(*=======================================================*)
	110: (* WT-Abfrage auf Beladeposition *)

		IF NOT e_station_vorher_in_abgegeben THEN
			a_station_vorher_out_angekommen := FALSE;
			bm_abfrage_wt_auf_beladepos := TRUE;
		END_IF

		(*-----------------------Weiterschaltbedingungen----------------------------*)
		IF e_wt_auf_beladepos THEN
			(* Ein WT ist anwesend zum rausschicken *)
			IF NOT ST_WT_Transport_Abgabe.e_wt_auf_abgabepos THEN
				(* Erst wenn kein Stau vorhanden ist, dann wird der WT weiter gelassen *)
				fb_state_entry.i16_next_step := 120;
			END_IF
		ELSE
			fb_state_entry.i16_next_step := 140;
		END_IF

		IF fb_state_entry.X THEN
			bm_abfrage_wt_auf_beladepos := FALSE;
			st_ctrl_out.b_kontroller_start := FALSE;
		END_IF

(*=======================================================*)
	120: (* WT-Zentrierer und Stopper einfahren *)
		IF fb_state_entry.E THEN
			zyl_wt_stopper_tisch.st_ctrl.in.b_einfahren := TRUE;
			zyl_wt_zentrierer_tisch.st_ctrl.in.b_einfahren := TRUE;
			fb_Zentrierer_einfahren(b_start:= TRUE, t_zeit=> );
			fb_Tisch_WechselZeit(b_start:=TRUE , t_zeit=> );
			pm_traegerwechselzeit := FALSE;
		END_IF

		IF 	zyl_wt_zentrierer_tisch.st_ctrl.out.b_eingefahren THEN
			fb_Zentrierer_einfahren(b_start:= FALSE, t_zeit=>t_Zentrierer_einfahren );
		END_IF

		(*-----------------------Weiterschaltbedingungen----------------------------*)
		IF zyl_wt_stopper_tisch.st_ctrl.out.b_eingefahren AND zyl_wt_zentrierer_tisch.st_ctrl.out.b_eingefahren THEN
			zyl_wt_stopper_tisch.st_ctrl.in.b_einfahren := FALSE;
			zyl_wt_zentrierer_tisch.st_ctrl.in.b_einfahren := FALSE;
			fb_state_entry.i16_next_step := 130;
		END_IF

(*=======================================================*)
	130: (* WT fährt von Bestücktisch heraus *)
		IF fb_state_entry.E THEN
			fb_ton_uez.PT := t#5s;
 			fb_ton_uez.IN := TRUE;
			st_ctrl_out.b_kontroller_start := TRUE;
		END_IF

		(*-----------------------Weiterschaltbedingungen----------------------------*)
		IF fb_r_trig_beladepos_verlassen.Q THEN
			fb_ton_uez.IN := FALSE;
			st_ctrl_out.b_kontroller_start := FALSE;
			IF	gst_datensatz.st_md.i16_WdhTouchProbe = 0 THEN
				fb_state_entry.i16_next_step := 144;
			ELSE
				fb_state_entry.i16_next_step := 140;
			END_IF
		ELSIF fb_ton_uez.Q THEN
			sm_wt_hat_beladepos_nicht_verlassen := TRUE;
			fb_state_entry.i16_next_step := FEHLER;
		END_IF

(*=======================================================*)
	140: (* Starte Touchprobe => kann immer gestartet werden. Wenn kein Taster eingebaut ist, wird gleich wieder fertig gemeldet*)
		IF fb_state_entry.E THEN
			ST_TouchProbe.st_ctrl_in.b_start := TRUE;
		END_IF

		(*-----------------------Weiterschaltbedingungen----------------------------*)
		IF	ST_TouchProbe.st_ctrl_out.b_busy THEN
			fb_state_entry.i16_next_step := 142;
		END_IF

(*=======================================================*)
	142: (* Warte auf fertig*)

		(*-----------------------Weiterschaltbedingungen----------------------------*)
		IF	ST_TouchProbe.st_ctrl_out.b_fertig THEN
			fb_state_entry.i16_next_step := 144;
		END_IF

(*=======================================================*)
	144: (* Stopper in Simulation nicht ausfahren  und  WT-Zentrierer einfahren *)
		IF fb_state_entry.E THEN
			zyl_wt_stopper_tisch.st_ctrl.in.b_ausfahren := TRUE;
			zyl_wt_zentrierer_tisch.st_ctrl.in.b_einfahren := TRUE;
		END_IF

		(*-----------------------Weiterschaltbedingungen----------------------------*)
		IF 	zyl_wt_stopper_tisch.st_ctrl.out.b_ausgefahren AND
			zyl_wt_zentrierer_tisch.st_ctrl.out.b_eingefahren
			THEN
				zyl_wt_stopper_tisch.st_ctrl.in.b_ausfahren := FALSE;
				zyl_wt_zentrierer_tisch.st_ctrl.in.b_einfahren := FALSE;
				fb_Tisch_WechselZeit(b_start:=FALSE , t_zeit=>t_tischwechselzeit );
				pm_traegerwechselzeit := t_tischwechselzeit > gst_datensatz.st_md.t_max_tischwechselzeit AND gst_datensatz.st_md.t_max_tischwechselzeit <> INT_TO_TIME(0);
				fb_state_entry.i16_next_step := 150;
		END_IF

(*=======================================================*)
	150: (* Warte auf Anforderung von vorheriger Station *)
		IF fb_state_entry.E THEN
			bm_warte_anforderung := TRUE;
		END_IF

		(*-----------------------Weiterschaltbedingungen----------------------------*)
		IF e_station_vorher_in_anforderung AND NOT e_wt_auf_beladepos THEN
			a_station_vorher_out_angekommen := FALSE;
			a_station_vorher_out_erlaubnis := TRUE;
			st_ctrl_out.b_kontroller_start := TRUE;
			bm_warte_anforderung := FALSE;
			fb_state_entry.i16_next_step := 160;
		END_IF

(*=======================================================*)
	160: (* Warte bis angekommen an Tisch-Stopper *)
		IF fb_state_entry.E THEN
			bm_warte_auf_wt_an_stopper := TRUE;
		END_IF

		IF e_wt_im_aktionsfeld AND NOT fb_ton_wz.Q THEN
			fb_ton_wz.PT := t#3s;
			fb_ton_wz.IN := TRUE;
		END_IF

		(*Kontroller neu starten wenn das Förderband zwischenzeitlich abgeschaltet hat*)
		IF 	e_station_vorher_in_abgegeben AND NOT ST_WT_Transport_Kontroller.a_foerderband_wt_transport THEN
			st_ctrl_out.b_kontroller_start := TRUE;
		ELSE
			st_ctrl_out.b_kontroller_start := FALSE;
		END_IF

		(*-----------------------Weiterschaltbedingungen----------------------------*)
		(* Auf das Kommando "e_station_vorher_in_abgegeben" wird nicht gewartet,
		da auch mal ein WT nach einer Störung so aus der vorherigen Station kommen kann. *)
		IF fb_ton_wt_auf_beladepos.Q THEN
			st_ctrl_out.b_kontroller_start := FALSE;
			a_station_vorher_out_erlaubnis := FALSE;
			a_station_vorher_out_angekommen := TRUE;
			bm_warte_auf_wt_an_stopper := FALSE;
			fb_ton_wz.IN := FALSE;
			fb_state_entry.i16_next_step := 170;
		END_IF

		(*Abfrage auf Sensorfehler des Beladepositionssensors *)
		IF e_wt_im_aktionsfeld AND NOT e_wt_auf_beladepos AND fb_ton_wz.Q THEN
			sm_sensorfehler_beladepos := TRUE;
			fb_state_entry.i16_next_step := FEHLER;
		END_IF

(*=======================================================*)
	170: (* WT-Zentrierer ausfahren *)
		IF fb_state_entry.E THEN
			zyl_wt_zentrierer_tisch.st_ctrl.in.b_ausfahren := TRUE;
			fb_Zentrierer_ausfahren(b_start:= TRUE, t_zeit=> );
		END_IF

		(*-----------------------Weiterschaltbedingungen----------------------------*)
		IF zyl_wt_zentrierer_tisch.st_ctrl.out.b_ausgefahren AND
			NOT ST_TippTasten.b_einfaedeln_aktiv AND
			(NOT ST_Virtuelle_Masterachse.b_merker_bandende_links  OR
 			NOT ST_Virtuelle_Masterachse.b_merker_bandende_rechts) THEN
			zyl_wt_zentrierer_tisch.st_ctrl.in.b_ausfahren := FALSE;
			fb_Zentrierer_ausfahren(b_start:= FALSE, t_zeit=> t_Zentrierer_ausfahren);
			zyl_wt_zentrierer_tisch.st_ctrl.in.b_ausfahren := FALSE;
			IF st_config.b_station_in_simulation THEN
				(* WT-Transport ist in Simulation und deshalb wird der WT ohne zu Bestücken weiter gefahren *)
				fb_state_entry.i16_next_step := BEREIT;
			ELSE
				fb_state_entry.i16_next_step := 190;
			END_IF
		END_IF

(*=======================================================*)
	190: (* WT-Tag mit RFID-Lesegerät abfragen *)
		IF fb_state_entry.E THEN
			fb_ton_wz.PT := t#100ms;
			fb_ton_wz.IN := TRUE;
		END_IF

		(*-----------------------Weiterschaltbedingungen----------------------------*)
		IF fb_ton_wz.Q THEN
			IF e_wt_im_aktionsfeld THEN
				(* Tag auslesen *)
				fb_state_entry.i16_next_step := 240;
			ELSE
				(* Kein Tag auf WT *)
				sm_wt_hat_kein_tag := TRUE;
				fb_state_entry.i16_next_step := FEHLER;
			END_IF
		END_IF

		IF fb_state_entry.X THEN
			fb_ton_wz.IN := FALSE;
		END_IF

(*=======================================================*)
	240: (* Starte Z-Achse *)
		IF fb_state_entry.E THEN
			axis_z_achse.st_ctrl.in.b_start := TRUE;
			st_ctrl_out.b_kontroller_start := TRUE;
			(*Zeitmessung Trägerwechsel stoppen und ausgeben*)
			fb_WT_WechselZeit(b_start:=FALSE , t_zeit=>t_WT_WechselZeit );
			(*Zeitmessung Bestückvorgang starten*)
			fb_Zentrierer_ausfahren(b_start:= FALSE, t_zeit=>t_Zentrierer_ausfahren );
		END_IF

		(*-----------------------Weiterschaltbedingungen----------------------------*)
		IF axis_z_achse.st_ctrl.out.b_fertig AND NOT fb_state_entry.E THEN
			axis_z_achse.st_ctrl.in.b_start := FALSE;
			st_ctrl_out.b_kontroller_start := FALSE;
			stueckzahlen.st_ctrl.in.b_gutteil_produziert := TRUE;
			(*Zeitmessung Trägerwechsel starten*)
			fb_WT_WechselZeit(b_start:=TRUE , t_zeit=> );
			(*Zeitmessung zusammenfassen*)
			t_bestueckzeit:=ST_Z_Achse.t_Bestueckung;
			t_traegerwechselzeit:=t_WT_WechselZeit + ST_Z_Achse.t_Z_Achse_einfahren + ST_Z_Achse.t_Z_Achse_ausfahren;
			t_komplett_zyklus:= t_traegerwechselzeit + t_bestueckzeit;
			fb_state_entry.i16_next_step := BEREIT;
		END_IF

		IF fb_state_entry.X THEN
			gst_datensatz.st_md.produzierte_Stecker := gst_datensatz.st_md.produzierte_Stecker + 1;
		END_IF

(*=======================================================*)
	500: (* Warte bis angekommen an Stopper *)
		IF fb_state_entry.E THEN
			bm_warte_auf_wt_an_stopper := TRUE;
		END_IF

		IF e_wt_im_aktionsfeld AND NOT fb_ton_wz.Q THEN
			fb_ton_wz.PT := t#3s;
			fb_ton_wz.IN := TRUE;
		END_IF

		(*-----------------------Weiterschaltbedingungen----------------------------*)
		IF fb_ton_wt_auf_beladepos.Q THEN
			fb_ton_wz.IN := FALSE;
			fb_state_entry.i16_next_step := 510;
		END_IF

		(*Abfrage auf Sensorfehler des Beladepositionssensors *)
		IF e_wt_im_aktionsfeld AND NOT e_wt_auf_beladepos AND fb_ton_wz.Q THEN
			sm_sensorfehler_beladepos := TRUE;
			fb_state_entry.i16_next_step := FEHLER;
		END_IF

(*=======================================================*)
	510: (* WT-Zentrierer ausfahren *)
		IF fb_state_entry.E THEN
			zyl_wt_zentrierer_tisch.st_ctrl.in.b_ausfahren := TRUE;
		END_IF

		(*-----------------------Weiterschaltbedingungen----------------------------*)
		IF zyl_wt_zentrierer_tisch.st_ctrl.out.b_ausgefahren  THEN
			zyl_wt_zentrierer_tisch.st_ctrl.in.b_ausfahren := FALSE;
			fb_state_entry.i16_next_step := 520;
		END_IF

(*=======================================================*)
	520:	(* Produktion ohne aktiven WT Transport *)
		IF fb_state_entry.E THEN
			axis_z_achse.st_ctrl.in.b_start := TRUE;
		END_IF

		(*-----------------------Weiterschaltbedingungen----------------------------*)
		IF axis_z_achse.st_ctrl.out.b_fertig AND NOT fb_state_entry.E THEN
			axis_z_achse.st_ctrl.in.b_start := FALSE;
			stueckzahlen.st_ctrl.in.b_gutteil_produziert := TRUE;
			IF NOT b_Dauertest_Achsen THEN
				fb_state_entry.i16_next_step := BEREIT;
			ELSE
				(* zum Testen der Achsen nach Tausch, Bestückbild "Becherspucken", WKZ ausgebaut, Vorschubkontrolle abeschaltet,
				Bit muss von Programmierer geforct werden, zum Beenden Schlüsselschalter auf HAND und Zelle neu starten *)
				fb_state_entry.i16_next_step := 500;	(* Dauertest *)
			END_IF
		END_IF

		IF fb_state_entry.X AND NOT b_Dauertest_Achsen THEN
			gst_datensatz.st_md.produzierte_Stecker := gst_datensatz.st_md.produzierte_Stecker + 1;
		END_IF

(*=======================================================*)
	FEHLER:
		IF fb_state_entry.E THEN
			st_ctrl_out.b_fehler := TRUE;
			fb_ton_quitt.IN := FALSE;
			zyl_wt_zentrierer_tisch.st_ctrl.in.b_quittieren := FALSE;
			zyl_wt_stopper_tisch.st_ctrl.in.b_quittieren := FALSE;

			a_station_vorher_out_erlaubnis := FALSE;
			a_station_vorher_out_angekommen := FALSE;

			st_ctrl_out.b_kontroller_start := FALSE;

			(*ST_Markiere_WT_NIO();*)
		END_IF

		(*-----------------------Weiterschaltbedingungen----------------------------*)
		IF st_ctrl_in.b_quitt AND NOT fb_state_entry.E THEN
			st_ctrl_out.b_fehler := FALSE;
			zyl_wt_zentrierer_tisch.st_ctrl.in.b_quittieren := TRUE;
			zyl_wt_stopper_tisch.st_ctrl.in.b_quittieren := TRUE;
			fb_ton_quitt.IN := TRUE;
		END_IF

		IF fb_ton_quitt.Q THEN
			fb_ton_quitt.IN := FALSE;
			fb_state_entry.i16_next_step := INIT;
		END_IF

(*=======================================================*)
	STOP:
		IF fb_state_entry.E THEN
			fb_ton_quitt.IN := FALSE;
			st_ctrl_out.b_kontroller_start := FALSE;
			zyl_wt_zentrierer_tisch.st_ctrl.in.b_quittieren := FALSE;
			zyl_wt_stopper_tisch.st_ctrl.in.b_quittieren := FALSE;
			a_station_vorher_out_erlaubnis := FALSE;
			a_station_vorher_out_angekommen := FALSE;
			(*ST_Markiere_WT_NIO();*)
		END_IF

		(*-----------------------Weiterschaltbedingungen----------------------------*)
		IF st_ctrl_in.b_quitt AND NOT fb_state_entry.E THEN
			fb_ton_quitt.IN := TRUE;
			zyl_wt_zentrierer_tisch.st_ctrl.in.b_quittieren := TRUE;
			zyl_wt_stopper_tisch.st_ctrl.in.b_quittieren := TRUE;
		END_IF

		IF fb_ton_quitt.Q THEN
			fb_ton_quitt.IN := FALSE;
			fb_state_entry.i16_next_step := INIT;
		END_IF
END_CASE

fb_state_entry(
	i16_next_step:= ,
	i16_pos:= 2,
	s_debugtext:= ,
	E=> ,
	X=> ,
	i16_step=> ,
	i16_last_step=> );

fb_ton_abfrage_wt_auf_beladepos (IN:=bm_abfrage_wt_auf_beladepos,PT:=t#30s);
fb_ton_warte_anforderung (IN:=bm_warte_anforderung,PT:=t#30s);
fb_ton_warte_auf_wt_an_stopper (IN:=bm_warte_auf_wt_an_stopper,PT:=t#30s);

IF st_config.b_config_fertig THEN
	(* Fehlermeldungen ab dem Startindex in das globale Störmeldungsarray schreiben *)
	garr_stoermeldungen[st_config.i16_meld_startindex + 0] := sm_wt_hat_beladepos_nicht_verlassen;
	garr_stoermeldungen[st_config.i16_meld_startindex + 1] := sm_tagnummer_ungueltig;
	garr_stoermeldungen[st_config.i16_meld_startindex + 2] := sm_wt_hat_kein_tag;
	garr_stoermeldungen[st_config.i16_meld_startindex + 3] := FALSE;
	garr_stoermeldungen[st_config.i16_meld_startindex + 4] := sm_sensorfehler_beladepos;
	garr_stoermeldungen[st_config.i16_meld_startindex + 5] := sm_tagreader_nicht_fertig;
	garr_stoermeldungen[st_config.i16_meld_startindex + 6] := sm_wt_zu_frueh_in_zelle;
	garr_stoermeldungen[st_config.i16_meld_startindex + 7] := sm_keine_bandfreigabe;
	garr_stoermeldungen[st_config.i16_meld_startindex + 8] := FALSE;
	garr_stoermeldungen[st_config.i16_meld_startindex + 9] := FALSE;
	garr_stoermeldungen[st_config.i16_meld_startindex + 10] := FALSE;
	garr_stoermeldungen[st_config.i16_meld_startindex + 11] := FALSE;
	garr_stoermeldungen[st_config.i16_meld_startindex + 12] := FALSE;
	garr_stoermeldungen[st_config.i16_meld_startindex + 13] := FALSE;
	garr_stoermeldungen[st_config.i16_meld_startindex + 14] := FALSE;
	garr_stoermeldungen[st_config.i16_meld_startindex + 15] := FALSE;
	garr_stoermeldungen[st_config.i16_meld_startindex + 16] := FALSE;
	garr_stoermeldungen[st_config.i16_meld_startindex + 17] := FALSE;
	garr_stoermeldungen[st_config.i16_meld_startindex + 18] := FALSE;
	garr_stoermeldungen[st_config.i16_meld_startindex + 19] := FALSE;
	
	garr_betriebsmeldungen[st_config.i16_meld_startindex + 0] := fb_ton_abfrage_wt_auf_beladepos.Q;
	garr_betriebsmeldungen[st_config.i16_meld_startindex + 1] := fb_ton_warte_anforderung.Q;
	garr_betriebsmeldungen[st_config.i16_meld_startindex + 2] := fb_ton_warte_auf_wt_an_stopper.Q;
	garr_betriebsmeldungen[st_config.i16_meld_startindex + 3] := FALSE;
	garr_betriebsmeldungen[st_config.i16_meld_startindex + 4] := FALSE;
	garr_betriebsmeldungen[st_config.i16_meld_startindex + 5] := FALSE;
	garr_betriebsmeldungen[st_config.i16_meld_startindex + 6] := FALSE;
	garr_betriebsmeldungen[st_config.i16_meld_startindex + 7] := FALSE;
	garr_betriebsmeldungen[st_config.i16_meld_startindex + 8] := FALSE;
	garr_betriebsmeldungen[st_config.i16_meld_startindex + 9] := FALSE;
	garr_betriebsmeldungen[st_config.i16_meld_startindex + 10] := FALSE;
	garr_betriebsmeldungen[st_config.i16_meld_startindex + 11] := FALSE;
	garr_betriebsmeldungen[st_config.i16_meld_startindex + 12] := FALSE;
	garr_betriebsmeldungen[st_config.i16_meld_startindex + 13] := FALSE;
	garr_betriebsmeldungen[st_config.i16_meld_startindex + 14] := FALSE;
	garr_betriebsmeldungen[st_config.i16_meld_startindex + 15] := FALSE;
	garr_betriebsmeldungen[st_config.i16_meld_startindex + 16] := FALSE;
	garr_betriebsmeldungen[st_config.i16_meld_startindex + 17] := FALSE;
	garr_betriebsmeldungen[st_config.i16_meld_startindex + 18] := FALSE;
	garr_betriebsmeldungen[st_config.i16_meld_startindex + 19] := FALSE;
END_IF
END_PROGRAM

(* POU Gemeinsamkeiten17xx/WT Transport/ST_WT_Transport_Kontroller, ST *)
PROGRAM ST_WT_Transport_Kontroller
VAR_INPUT
	st_config								: struct_config;
	st_ctrl_in								: struct_ctrl_in;
END_VAR
VAR_IN_OUT
	st_visu								: struct_visu;
END_VAR
VAR_OUTPUT
	st_ctrl_out							: struct_ctrl_out;
END_VAR
VAR
	fb_ton_uez							: TON;
	fb_ton_wz							: TON;
	fb_ton_quitt							: TON;
	fb_ton_stausensor						: TON;
	fb_ton_wz_nachlauf_fb_oben			: TON;
	fb_ton_wz_nachlauf_fb_unten			: TON;
	fb_ton_wz_foerderband_stauzeit			: TON;
	fb_ton_ueberstrom_foerderbaender		: TON;
	fb_r_trig_beladen_start_fb				: R_TRIG;
	fb_r_trig_beladen_1700_start_fb			: R_TRIG;
	fb_r_trig_beladen_wartepos_1700_start_fb	: R_TRIG;
	fb_r_trig_abgabe_start_fb				: R_TRIG;
	fb_r_trig_wartepos_start_fb				: R_TRIG;
	fb_r_trig_start_foerderband				: R_TRIG;
	fb_r_trig_eigenstart_foerderband			: R_TRIG;
	fb_r_trig_hublift						: R_TRIG;
	fb_state_entry							: ST_StateEntry;
	t_foerderband_nachlaufzeit				: TIME := t#10m;
	t_foerderband_stauzeit					: TIME := t#1s;
	b_eigenstart_foerderband				: BOOL := FALSE;
	b_ibn_rundlauf_tipptaste				: BOOL := FALSE;	(* Merker für endlos Lauf und keinen WT-Transport - wird nur im PLC händisch gesetzt *)
	i									: DINT := 0;

	sm_stau_auf_ruecktransport				: BOOL := FALSE;
	sm_ueberstrom_foerderbaender			: BOOL := FALSE;

	bm_einzelfertigung_nach_bandwechsel	: BOOL := FALSE;
	e_stausensor_wt_ruecktransport			AT %I* : BOOL;
	a_foerderband_wt_transport				AT %Q* : BOOL;
	a_foerderband_wt_ruecktransport		AT %Q* : BOOL;
	e_ueberstrom_foerderbaender			AT %I* : BOOL;
END_VAR
(* Zeiten *)
fb_ton_uez(IN:= , PT:= , Q=>  , ET=> );
fb_ton_wz(IN:= , PT:= , Q=> , ET=> );
fb_ton_quitt(IN:= , PT:= t#150ms, Q=> , ET=> );



(*Trigger*)
CASE gst_datensatz.st_md.i16_typ_zelle OF
	KEINE_ZELLE:
		;

	BESTUECKZELLE_1700, RASTERFOLIE:
		IF NOT gst_datensatz.st_md.b_anwahl_transport_achse THEN
			fb_r_trig_beladen_start_fb(CLK:= wt_transport_beladen.st_ctrl.out.b_kontroller_start, Q=> );
			fb_ton_wz_foerderband_stauzeit(IN:=  ST_WT_Transport_Beladen.e_wt_auf_beladepos AND ST_WT_Transport_Abgabe.e_wt_auf_abgabepos, PT:= t_foerderband_stauzeit, Q=> , ET=> );
		ELSE
			fb_r_trig_beladen_1700_start_fb(CLK:= wt_transport_beladen_achse_1700.st_ctrl.out.b_kontroller_start, Q=> );
			fb_r_trig_beladen_wartepos_1700_start_fb(CLK:= wt_transport_warteposition_1700.st_ctrl.out.b_kontroller_start, Q=> );
			fb_ton_wz_foerderband_stauzeit(IN:= ST_WT_Transport_Warteposition_1700.e_wt_auf_wartepos_1700 AND ST_WT_Transport_Abgabe.e_wt_auf_abgabepos, PT:= t_foerderband_stauzeit, Q=> , ET=> );
		END_IF

	BESTUECKZELLE_1720:
		fb_r_trig_beladen_start_fb(CLK:= wt_transport_beladen_1720.st_ctrl.out.b_kontroller_start, Q=> );
		fb_r_trig_wartepos_start_fb(CLK:= wt_transport_warteposition_1720.st_ctrl.out.b_kontroller_start, Q=> );
		fb_ton_wz_foerderband_stauzeit(IN:=  ST_WT_Transport_Beladen_1720.e_wt_auf_beladepos AND ST_WT_Transport_Abgabe.e_wt_auf_abgabepos AND ST_WT_Transport_Warteposition_1720.e_wt_auf_wartepos , PT:= t_foerderband_stauzeit, Q=> , ET=> );
END_CASE

fb_r_trig_abgabe_start_fb(CLK:= wt_transport_abgabe.st_ctrl.out.b_kontroller_start, Q=> );
fb_r_trig_start_foerderband(CLK:= st_visu.b_start_foerderband, Q=> );
fb_r_trig_eigenstart_foerderband(CLK:= b_eigenstart_foerderband, Q=> );
fb_r_trig_hublift(CLK:= hublift_links.st_ctrl.out.b_kontroller_start, Q=> );
fb_ton_ueberstrom_foerderbaender(IN:=NOT e_ueberstrom_foerderbaender  , PT:= t#200ms, Q=> , ET=> );

(* =====Ansteuerung Förderbänder===== *)
fb_ton_stausensor(IN:= e_stausensor_wt_ruecktransport AND
					NOT st_visu.b_start_foerderband AND
					NOT fb_r_trig_beladen_start_fb.Q AND
					NOT fb_r_trig_wartepos_start_fb.Q AND
					NOT fb_r_trig_beladen_1700_start_fb.Q AND
					NOT fb_r_trig_beladen_wartepos_1700_start_fb.Q

					, PT:= t#5s, Q=> , ET=> );

fb_ton_wz_nachlauf_fb_oben(IN:= , PT:= t_foerderband_nachlaufzeit, Q=> , ET=> );
fb_ton_wz_nachlauf_fb_unten(IN:= , PT:= t_foerderband_nachlaufzeit, Q=> , ET=> );

(* ===Zeit nachtriggern=== *)
(* Förderband oben *)
IF 	fb_r_trig_beladen_start_fb.Q OR
	fb_r_trig_abgabe_start_fb.Q OR
	fb_r_trig_wartepos_start_fb.Q OR
	 fb_r_trig_beladen_1700_start_fb.Q OR
	fb_r_trig_beladen_wartepos_1700_start_fb.Q OR
	fb_r_trig_hublift.Q
	THEN
		fb_ton_wz_nachlauf_fb_oben(IN:= FALSE, PT:= t_foerderband_nachlaufzeit, Q=> , ET=> );
END_IF
(* Förderband unten *)
IF 	fb_r_trig_beladen_start_fb.Q OR
	fb_r_trig_abgabe_start_fb.Q OR
	fb_r_trig_wartepos_start_fb.Q OR
	 fb_r_trig_beladen_1700_start_fb.Q OR
	fb_r_trig_beladen_wartepos_1700_start_fb.Q OR
	fb_r_trig_start_foerderband.Q
	THEN
		fb_ton_wz_nachlauf_fb_unten(IN:= FALSE, PT:= t_foerderband_nachlaufzeit, Q=> , ET=> );
END_IF

(* ===Ansteuerung=== *)
(* Förderband oben *)
IF 	ST_Safetyprogramm.se_steuerung_ein AND ST_Safetyprogramm.se_ba_mit_bedingungen AND
	(st_config.b_station_aktiv  OR st_config.b_station_in_simulation)
	THEN
		IF 	fb_r_trig_beladen_start_fb.Q OR
			fb_r_trig_abgabe_start_fb.Q OR
			fb_r_trig_wartepos_start_fb.Q OR
			fb_r_trig_eigenstart_foerderband.Q OR
			 fb_r_trig_beladen_1700_start_fb.Q OR
			fb_r_trig_beladen_wartepos_1700_start_fb.Q OR
			fb_r_trig_hublift.Q
			 THEN
				a_foerderband_wt_transport := TRUE;
				fb_ton_wz_nachlauf_fb_oben(IN:= TRUE, PT:= t_foerderband_nachlaufzeit, Q=> , ET=> );
				fb_ton_wz_foerderband_stauzeit(IN:= FALSE, PT:= t_foerderband_nachlaufzeit, Q=> , ET=> );
		ELSE
			IF fb_ton_wz_nachlauf_fb_oben.Q OR fb_ton_wz_foerderband_stauzeit.Q THEN
				a_foerderband_wt_transport := FALSE;
				fb_ton_wz_nachlauf_fb_oben(IN:= FALSE, PT:= t_foerderband_nachlaufzeit, Q=> , ET=> );
			END_IF
		END_IF
ELSE
	fb_ton_wz_nachlauf_fb_unten.IN := FALSE;
	a_foerderband_wt_transport := FALSE;
END_IF

(* Förderband unten *)
(* Funktionsweise:
Bei Anforderung von vorheriger Station an das Fb oben wird ebenso das Fb unten gestartet. Somit setzt sich die Kette wieder Bewegung. 
Mit Handstart kann die Anlage in Richtung BEHR-Zelle entleert werden, ohne dass neue WTs oben kommen. *)
IF 	ST_Safetyprogramm.se_steuerung_ein AND ST_Safetyprogramm.se_ba_mit_bedingungen AND
	(st_config.b_station_aktiv  OR st_config.b_station_in_simulation)
	THEN
		IF 	fb_r_trig_beladen_start_fb.Q OR
			fb_r_trig_abgabe_start_fb.Q OR
			fb_r_trig_wartepos_start_fb.Q OR
			fb_r_trig_start_foerderband.Q OR
			fb_r_trig_beladen_1700_start_fb.Q OR
			fb_r_trig_beladen_wartepos_1700_start_fb.Q OR
			fb_r_trig_eigenstart_foerderband.Q
			THEN
				a_foerderband_wt_ruecktransport := TRUE;
				fb_ton_wz_nachlauf_fb_unten(IN:= TRUE, PT:= t_foerderband_nachlaufzeit, Q=> , ET=> );
		ELSE
			IF fb_ton_wz_nachlauf_fb_unten.Q OR fb_ton_stausensor.Q THEN
				a_foerderband_wt_ruecktransport := FALSE;
				fb_ton_wz_nachlauf_fb_unten(IN:= FALSE, PT:= t_foerderband_nachlaufzeit, Q=> , ET=> );
			END_IF
		END_IF
ELSE
	fb_ton_wz_nachlauf_fb_unten.IN := FALSE;
	a_foerderband_wt_ruecktransport := FALSE;
END_IF


(* =================================Toplevel=================================== *)
IF fb_state_entry.i16_next_step > INIT AND fb_state_entry.i16_next_step < FEHLER THEN
	IF fb_state_entry.i16_next_step < STOP THEN
		IF st_ctrl_in.b_stop THEN
			fb_state_entry.i16_next_step := STOP;
		END_IF
	END_IF

	(* Allgemeine Fehler *)
	IF	wt_transport_beladen.st_ctrl.out.b_fehler OR
		wt_transport_beladen_achse_1700.st_ctrl.out.b_fehler OR
		wt_transport_beladen_1720.st_ctrl.out.b_fehler
		THEN
			fb_state_entry.i16_next_step := FEHLER;
	END_IF
END_IF

(* ==================================Schrittkette================================ *)
fb_state_entry(
	i16_next_step:= ,
	i16_pos:= 1,
	s_debugtext:= ,
	E=> ,
	X=> ,
	i16_step=> ,
	i16_last_step=> );

CASE fb_state_entry.i16_step OF
(*=======================================================*)
	INIT_OBJ:
		IF st_config.b_config_fertig THEN
			fb_state_entry.i16_next_step := INIT;
		END_IF

(*=======================================================*)
	INIT:
		IF fb_state_entry.E THEN
			fb_ton_wz.IN := FALSE;
			fb_ton_uez.IN := FALSE;
			fb_ton_quitt.IN := FALSE;
			st_ctrl_out.b_fehler := FALSE;
			st_ctrl_out.b_bereit := FALSE;
			st_ctrl_out.b_fertig := FALSE;
			sm_stau_auf_ruecktransport := FALSE;
			sm_ueberstrom_foerderbaender := FALSE;
			bm_einzelfertigung_nach_bandwechsel := FALSE;

			wt_transport_beladen.st_ctrl.in.b_init := FALSE;
			wt_transport_abgabe.st_ctrl.in.b_init := FALSE;
			wt_transport_warteposition_1700.st_ctrl.in.b_init := FALSE;
			wt_transport_beladen_achse_1700.st_ctrl.in.b_init := FALSE;
			wt_transport_warteposition_1720.st_ctrl.in.b_init := FALSE;
			wt_transport_beladen_1720.st_ctrl.in.b_init := FALSE;
			wt_transport_beladen.st_ctrl.in.b_start := FALSE;
			wt_transport_abgabe.st_ctrl.in.b_start := FALSE;
			wt_transport_warteposition_1700.st_ctrl.in.b_start := FALSE;
			wt_transport_beladen_achse_1700.st_ctrl.in.b_start := FALSE;
			wt_transport_warteposition_1720.st_ctrl.in.b_start := FALSE;
			wt_transport_beladen_1720.st_ctrl.in.b_start := FALSE;

			gb_nach_bawe_einzelfertigung := FALSE;
		END_IF

		(*-----------------------Weiterschaltbedingungen----------------------------*)
		IF st_ctrl_in.b_init THEN
			EtherCatDiag[1].st_ctrl_in.b_quitt := TRUE;
			EtherCatDiag[2].st_ctrl_in.b_quitt := TRUE;
			EtherCatDiag[3].st_ctrl_in.b_quitt := TRUE;
			EtherCatDiag[4].st_ctrl_in.b_quitt := TRUE;
			wt_transport_beladen.st_ctrl.in.b_quitt := FALSE;
			wt_transport_abgabe.st_ctrl.in.b_quitt := FALSE;
			wt_transport_warteposition_1700.st_ctrl.in.b_quitt := FALSE;
			wt_transport_beladen_achse_1700.st_ctrl.in.b_quitt := FALSE;
			wt_transport_warteposition_1720.st_ctrl.in.b_quitt := FALSE;
			wt_transport_beladen_1720.st_ctrl.in.b_quitt := FALSE;
			fb_ton_ueberstrom_foerderbaender.IN := FALSE;
			fb_state_entry.i16_next_step := 20;
		END_IF

(*=======================================================*)
	20: (* Initialisierung Subkomponenten *)
		CASE gst_datensatz.st_md.i16_typ_zelle OF
			KEINE_ZELLE:
				;

			BESTUECKZELLE_1700, RASTERFOLIE:
				IF fb_state_entry.E THEN
					IF gst_datensatz.st_md.b_anwahl_transport_achse THEN
						wt_transport_beladen_achse_1700.st_ctrl.in.b_init := TRUE;
						wt_transport_warteposition_1700.st_ctrl.in.b_init := TRUE;
					ELSE
						wt_transport_beladen.st_ctrl.in.b_init := TRUE;
					END_IF
					wt_transport_abgabe.st_ctrl.in.b_init := TRUE;
				END_IF

				(*-----------------------Weiterschaltbedingungen----------------------------*)
				IF gst_datensatz.st_md.b_anwahl_transport_achse THEN
					IF 	wt_transport_beladen_achse_1700.st_ctrl.out.b_bereit AND
						wt_transport_warteposition_1700.st_ctrl.out.b_bereit AND
						wt_transport_abgabe.st_ctrl.out.b_bereit THEN
						wt_transport_beladen_achse_1700.st_ctrl.in.b_init := FALSE;
						wt_transport_warteposition_1700.st_ctrl.in.b_init := FALSE;
						wt_transport_abgabe.st_ctrl.in.b_init := FALSE;
						fb_state_entry.i16_next_step := BEREIT;
					END_IF
				ELSE
					IF 	wt_transport_beladen.st_ctrl.out.b_bereit AND
						wt_transport_abgabe.st_ctrl.out.b_bereit THEN
						wt_transport_beladen.st_ctrl.in.b_init := FALSE;
						wt_transport_abgabe.st_ctrl.in.b_init := FALSE;
						fb_state_entry.i16_next_step := BEREIT;
					END_IF
				END_IF


			BESTUECKZELLE_1720:
				IF fb_state_entry.E THEN
					wt_transport_warteposition_1720.st_ctrl.in.b_init := TRUE;
					wt_transport_beladen_1720.st_ctrl.in.b_init := TRUE;
					wt_transport_abgabe.st_ctrl.in.b_init := TRUE;
				END_IF
		
				(*-----------------------Weiterschaltbedingungen----------------------------*)
				IF	wt_transport_warteposition_1720.st_ctrl.out.b_bereit AND
					wt_transport_beladen_1720.st_ctrl.out.b_bereit AND
					wt_transport_abgabe.st_ctrl.out.b_bereit
					THEN
						wt_transport_warteposition_1720.st_ctrl.in.b_init := FALSE;
						wt_transport_beladen_1720.st_ctrl.in.b_init := FALSE;
						wt_transport_abgabe.st_ctrl.in.b_init := FALSE;
						b_eigenstart_foerderband := TRUE;
						fb_state_entry.i16_next_step := BEREIT;
				END_IF
		END_CASE

		IF fb_state_entry.X THEN
			EtherCatDiag[1].st_ctrl_in.b_quitt := FALSE;
			EtherCatDiag[2].st_ctrl_in.b_quitt := FALSE;
			EtherCatDiag[3].st_ctrl_in.b_quitt := FALSE;
			EtherCatDiag[4].st_ctrl_in.b_quitt := FALSE;
		END_IF

(*=======================================================*)
	BEREIT:	(* WT-Stationen sind bereit für Annahme oder Abgabe *)
		IF fb_state_entry.E THEN
			st_ctrl_out.b_bereit := TRUE;
			st_ctrl_out.b_fertig := TRUE;
			b_eigenstart_foerderband := FALSE;
			bm_einzelfertigung_nach_bandwechsel := FALSE;
		END_IF

		(*-----------------------Weiterschaltbedingungen----------------------------*)
		CASE gst_datensatz.st_md.i16_typ_zelle OF
			KEINE_ZELLE:
				;
			RASTERFOLIE:
				IF st_config.b_station_aktiv  OR st_config.b_station_in_simulation THEN
					(* WT-Transport aktiv oder in Simulation *)
					(* Warte auf Start *)
					IF ST_TippTasten.r_trig_tippen.Q THEN
						st_ctrl_out.b_fertig := FALSE;
						wt_transport_beladen.st_ctrl.in.b_start := TRUE;
						wt_transport_abgabe.st_ctrl.in.b_start := TRUE;
						fb_state_entry.i16_next_step := 110;
					END_IF
				ELSE
					(* WT-Transport nicht aktiv  *)
					wt_transport_abgabe.st_ctrl.in.b_start := FALSE;
					(* Warte auf Start *)
					IF ST_TippTasten.r_trig_tippen.Q OR b_ibn_rundlauf_tipptaste THEN
						st_ctrl_out.b_fertig := FALSE;
						fb_state_entry.i16_next_step := 200;
					END_IF
				END_IF

			BESTUECKZELLE_1700:
				(* WT-Transport aktiv oder in Simulation *)
				IF st_config.b_station_aktiv  OR st_config.b_station_in_simulation THEN
					(* Warte auf Start von Visu bzw. Handbedienpult wenn kein Bandwechsel war *)
					IF ST_TippTasten.r_trig_tippen.Q THEN
						st_ctrl_out.b_fertig := FALSE;
						IF gst_datensatz.st_md.b_anwahl_transport_achse THEN
							wt_transport_beladen_achse_1700.st_ctrl.in.b_start := TRUE;
							wt_transport_warteposition_1700.st_ctrl.in.b_start := TRUE;
						ELSE
							wt_transport_beladen.st_ctrl.in.b_start := TRUE;
						END_IF
						wt_transport_abgabe.st_ctrl.in.b_start := TRUE;
						fb_state_entry.i16_next_step := 110;
					END_IF

				(* WT-Transport nicht aktiv  *)
				ELSE
					wt_transport_abgabe.st_ctrl.in.b_start := FALSE;
					(* Warte auf Start von Visu oder Handbedienpult *)
					IF ST_TippTasten.r_trig_tippen.Q OR b_ibn_rundlauf_tipptaste THEN
						st_ctrl_out.b_fertig := FALSE;
						bm_einzelfertigung_nach_bandwechsel := FALSE;
						fb_state_entry.i16_next_step := 200;
					END_IF
				END_IF

			BESTUECKZELLE_1720:
				IF st_config.b_station_aktiv  OR st_config.b_station_in_simulation THEN
					(* WT-Transport aktiv oder in Simulation *)
					(* Warte auf Start von Visu oder Handbedienpult *)
					IF ST_TippTasten.r_trig_tippen.Q THEN
						st_ctrl_out.b_fertig := FALSE;
						wt_transport_abgabe.st_ctrl.in.b_start := TRUE;
						wt_transport_warteposition_1720.st_ctrl.in.b_start := TRUE;
						wt_transport_beladen_1720.st_ctrl.in.b_start := TRUE;
						fb_state_entry.i16_next_step := 110;
					END_IF
				ELSE
					(* WT-Transport nicht aktiv  *)
					wt_transport_abgabe.st_ctrl.in.b_start := FALSE;
					wt_transport_warteposition_1720.st_ctrl.in.b_start := FALSE;
					(* Warte auf Start von Visu oder Handbedienpult *)
					IF ST_TippTasten.r_trig_tippen.Q OR b_ibn_rundlauf_tipptaste THEN
						st_ctrl_out.b_fertig := FALSE;
						fb_state_entry.i16_next_step := 200;
					END_IF
				END_IF

		END_CASE

(*=======================================================*)
	105: (* Wenn der Bediener nach einem Bandwechsel die niO Taste auf der Visu drückt, wird der WT als schlecht beschrieben *)
		IF fb_state_entry.E THEN
			(* WT  mit "nio" beschreiben *)
			ST_Markiere_WT_NIO();
		END_IF

		(*-----------------------Weiterschaltbedingungen----------------------------*)
		IF balluff_tag_reader.st_ctrl.out.b_fertig AND NOT fb_state_entry.E THEN
			balluff_tag_reader.st_ctrl.in.b_start_schreiben := FALSE;
			IF gst_datensatz.st_md.b_anwahl_transport_achse THEN
				wt_transport_beladen_achse_1700.st_ctrl.in.b_start := TRUE;
				wt_transport_warteposition_1700.st_ctrl.in.b_start := TRUE;
			ELSE
				wt_transport_beladen.st_ctrl.in.b_start := TRUE;
			END_IF
			wt_transport_abgabe.st_ctrl.in.b_start := TRUE;
			fb_state_entry.i16_next_step := 107;
		END_IF

(*=======================================================*)
	107: (* Anlage wird wieder in Einzelfertigung geschickt *)
		IF fb_state_entry.E THEN
			IF gst_datensatz.st_md.b_anwahl_transport_achse THEN
				wt_transport_beladen_achse_1700.st_ctrl.in.b_start := FALSE;
				wt_transport_warteposition_1700.st_ctrl.in.b_start := FALSE;
			ELSE
				wt_transport_beladen.st_ctrl.in.b_start := FALSE;
			END_IF
			wt_transport_abgabe.st_ctrl.in.b_start := FALSE;
		END_IF

		(*-----------------------Weiterschaltbedingungen----------------------------*)
		fb_state_entry.i16_next_step := 120;

(*=======================================================*)
	110:	(* Produktion: Anlage läuft im Verbund *)

		(*-----------------------Weiterschaltbedingungen----------------------------*)
		CASE gst_datensatz.st_md.i16_typ_zelle OF
			KEINE_ZELLE:
				;

			BESTUECKZELLE_1700:
				IF 	visu.b_einzelfertigung OR visu_hinten.out.b_einzelfertigung OR gb_nach_bawe_einzelfertigung OR bandspruehoeler.st_ctrl.out.b_einzelfertigung THEN
					IF gb_nach_bawe_einzelfertigung THEN
						bm_einzelfertigung_nach_bandwechsel := TRUE;
					END_IF
					IF gst_datensatz.st_md.b_anwahl_transport_achse THEN
						wt_transport_beladen_achse_1700.st_ctrl.in.b_start := FALSE;
						wt_transport_warteposition_1700.st_ctrl.in.b_start := FALSE;
					ELSE
						wt_transport_beladen.st_ctrl.in.b_start := FALSE;
					END_IF
					wt_transport_abgabe.st_ctrl.in.b_start := FALSE;
					gb_nach_bawe_einzelfertigung := FALSE;
					fb_state_entry.i16_next_step := 120;
				ELSIF 	hublift_links.st_ctrl.out.b_fehler OR
						hublift_rechts.st_ctrl.out.b_fehler OR
						(wt_transport_beladen.st_ctrl.out.b_fehler AND NOT gst_datensatz.st_md.b_anwahl_transport_achse) OR
						(wt_transport_beladen_achse_1700.st_ctrl.out.b_fehler AND gst_datensatz.st_md.b_anwahl_transport_achse) OR
						wt_transport_warteposition_1700.st_ctrl.out.b_fehler OR
						wt_transport_abgabe.st_ctrl.out.b_fehler OR
						EtherCatDiag[1].st_ctrl_out.b_fehler OR
						EtherCatDiag[2].st_ctrl_out.b_fehler OR
						EtherCatDiag[3].st_ctrl_out.b_fehler OR
						EtherCatDiag[4].st_ctrl_out.b_fehler OR
						fb_ton_ueberstrom_foerderbaender.Q THEN
						IF gst_datensatz.st_md.b_anwahl_transport_achse THEN
							wt_transport_beladen_achse_1700.st_ctrl.in.b_start := FALSE;
							wt_transport_warteposition_1700.st_ctrl.in.b_start := FALSE;
						ELSE
							wt_transport_beladen.st_ctrl.in.b_start := FALSE;
						END_IF
						wt_transport_abgabe.st_ctrl.in.b_start := FALSE;
						gb_nach_bawe_einzelfertigung := FALSE;
						fb_state_entry.i16_next_step := 130;
				END_IF

			BESTUECKZELLE_1720:
				IF visu.b_einzelfertigung OR visu_hinten.out.b_einzelfertigung OR gb_nach_bawe_einzelfertigung OR ST_WkzAbsicherung.st_ctrl_out.b_einzelfertigung OR bandspruehoeler.st_ctrl.out.b_einzelfertigung  THEN
					wt_transport_warteposition_1720.st_ctrl.in.b_start := FALSE;
					wt_transport_beladen_1720.st_ctrl.in.b_start := FALSE;
					wt_transport_abgabe.st_ctrl.in.b_start := FALSE;
					gb_nach_bawe_einzelfertigung := FALSE;
					fb_state_entry.i16_next_step := 120;
				ELSIF 	hublift_links.st_ctrl.out.b_fehler OR
						hublift_rechts.st_ctrl.out.b_fehler OR
						wt_transport_warteposition_1720.st_ctrl.out.b_fehler OR
						EtherCatDiag[1].st_ctrl_out.b_fehler OR
						EtherCatDiag[2].st_ctrl_out.b_fehler OR
						EtherCatDiag[3].st_ctrl_out.b_fehler OR
						EtherCatDiag[4].st_ctrl_out.b_fehler OR
						fb_ton_ueberstrom_foerderbaender.Q THEN
						wt_transport_warteposition_1720.st_ctrl.in.b_start := FALSE;
						wt_transport_beladen_1720.st_ctrl.in.b_start := FALSE;
						wt_transport_abgabe.st_ctrl.in.b_start := FALSE;
						gb_nach_bawe_einzelfertigung := FALSE;
						fb_state_entry.i16_next_step := 130;
				END_IF

			RASTERFOLIE:
				IF visu.b_einzelfertigung OR visu_hinten.out.b_einzelfertigung THEN
					wt_transport_beladen.st_ctrl.in.b_start := FALSE;
					wt_transport_abgabe.st_ctrl.in.b_start := FALSE;
					fb_state_entry.i16_next_step := 120;
				ELSIF 	hublift_links.st_ctrl.out.b_fehler OR
						hublift_rechts.st_ctrl.out.b_fehler OR
						wt_transport_abgabe.st_ctrl.out.b_fehler OR
						EtherCatDiag[1].st_ctrl_out.b_fehler OR
						EtherCatDiag[2].st_ctrl_out.b_fehler OR
						EtherCatDiag[3].st_ctrl_out.b_fehler OR
						EtherCatDiag[4].st_ctrl_out.b_fehler OR
						fb_ton_ueberstrom_foerderbaender.Q THEN
						wt_transport_beladen.st_ctrl.in.b_start := FALSE;
						wt_transport_abgabe.st_ctrl.in.b_start := FALSE;
						fb_state_entry.i16_next_step := 130;
				END_IF
		END_CASE

(*=======================================================*)
	120:	(* Produktion beenden, wenn WT fertig bestückt *)
		CASE gst_datensatz.st_md.i16_typ_zelle OF
			KEINE_ZELLE:
				;

			BESTUECKZELLE_1700, RASTERFOLIE:
			(*-----------------------Weiterschaltbedingungen----------------------------*)
				IF gst_datensatz.st_md.b_anwahl_transport_achse THEN
					IF wt_transport_beladen_achse_1700.st_ctrl.out.b_fertig THEN
						fb_state_entry.i16_next_step := BEREIT;
					END_IF
				ELSE
					IF wt_transport_beladen.st_ctrl.out.b_fertig THEN
						fb_state_entry.i16_next_step := BEREIT;
					END_IF
				END_IF

			BESTUECKZELLE_1720:
			(*-----------------------Weiterschaltbedingungen----------------------------*)
				IF wt_transport_beladen_1720.st_ctrl.out.b_fertig THEN
					fb_state_entry.i16_next_step := BEREIT;
				END_IF
		END_CASE

(*=======================================================*)
	130:	(* Produktion beenden, wenn WT fertig bestückt, dann FEHLER*)
		CASE gst_datensatz.st_md.i16_typ_zelle OF
			KEINE_ZELLE:
				;

			BESTUECKZELLE_1700, RASTERFOLIE:
			IF 	fb_ton_ueberstrom_foerderbaender.Q THEN
				sm_ueberstrom_foerderbaender := TRUE;
			END_IF
			(*-----------------------Weiterschaltbedingungen----------------------------*)
				IF gst_datensatz.st_md.b_anwahl_transport_achse THEN
					IF 	wt_transport_beladen_achse_1700.st_ctrl.out.b_fertig OR
						wt_transport_beladen_achse_1700.st_ctrl.out.b_fehler THEN
						fb_state_entry.i16_next_step := FEHLER;
					END_IF
				ELSE
					IF 	wt_transport_beladen.st_ctrl.out.b_fertig OR
						wt_transport_beladen.st_ctrl.out.b_fehler THEN
						fb_state_entry.i16_next_step := FEHLER;
					END_IF
				END_IF

			BESTUECKZELLE_1720:
			IF 	fb_ton_ueberstrom_foerderbaender.Q THEN
				sm_ueberstrom_foerderbaender := TRUE;
			END_IF
			(*-----------------------Weiterschaltbedingungen----------------------------*)
				IF wt_transport_beladen_1720.st_ctrl.out.b_fertig THEN
					fb_state_entry.i16_next_step := FEHLER;
				END_IF
		END_CASE

		IF fb_state_entry.E THEN
			fb_ton_ueberstrom_foerderbaender.IN := FALSE;
		END_IF
(*=======================================================*)
	200: (*Warten bis keine ander Produktions Meldung ansteht *)

		(*-----------------------Weiterschaltbedingungen----------------------------*)
		IF	TestAndSet(ST_Message_Produktion.LockFlag) THEN
			ST_Message_Produktion.ClearMessageLines();
			fb_state_entry.i16_next_step := 201;
		END_IF

(*=======================================================*)
	201:  (*Produktions Meldung*)
		Visu.MeldungProduktion.Color_R := 255;
		Visu.MeldungProduktion.Color_G := 0;
		Visu.MeldungProduktion.Color_B := 0;
		IF visu.s_akt_sprache = 'de' THEN
			Visu.MeldungProduktion.Name:='WT Transport nicht aktiviert. Weiter mit OK';
		ELSIF visu.s_akt_sprache = 'en' THEN
			Visu.MeldungProduktion.Name:='carrier transport deactivated. Confirm with OK';
		ELSIF visu.s_akt_sprache = 'cz' THEN
			Visu.MeldungProduktion.Name:='Transport WT deaktivovan. Potvrdte pres OK';
		END_IF
		Visu.MeldungProduktion.ShowMessage := TRUE;
		Visu.MeldungProduktion.Button1.sichtbar:=TRUE;	(*OK*)
		Visu.MeldungProduktion.Button1.Text:='Ok';
		Visu.MeldungProduktion.Button2.sichtbar:=TRUE;	(*Abbrechen*)
		Visu.MeldungProduktion.Button2.Text:='Abbrechen';

		(*-----------------------Weiterschaltbedingungen----------------------------*)
		fb_state_entry.i16_next_step := 202;

(*=======================================================*)
	202:  (*Warte auf OK*)

		(*-----------------------Weiterschaltbedingungen----------------------------*)
		IF Visu.MeldungProduktion.Button1.tasten THEN
			IF gst_datensatz.st_md.b_anwahl_transport_achse THEN
				wt_transport_beladen_achse_1700.st_ctrl.in.b_start := TRUE;
			ELSE
				wt_transport_beladen.st_ctrl.in.b_start := TRUE;
			END_IF
			wt_transport_beladen_1720.st_ctrl.in.b_start := TRUE;
			fb_state_entry.i16_next_step:=210;
		ELSIF Visu.MeldungProduktion.Button2.tasten THEN
			fb_state_entry.i16_next_step:=100;
		END_IF

(*=======================================================*)
	210:	(* Produktion: Anlage läuft im Singelbetrieb *)

		CASE gst_datensatz.st_md.i16_typ_zelle OF
			KEINE_ZELLE:
				;

			BESTUECKZELLE_1700, RASTERFOLIE:
			(*-----------------------Weiterschaltbedingungen----------------------------*)
				IF gst_datensatz.st_md.b_anwahl_transport_achse THEN
					IF wt_transport_beladen_achse_1700.st_ctrl.out.b_fertig THEN
						wt_transport_beladen_achse_1700.st_ctrl.in.b_start := FALSE;
						fb_state_entry.i16_next_step := BEREIT;
					END_IF
				ELSE
					IF wt_transport_beladen.st_ctrl.out.b_fertig THEN
						wt_transport_beladen.st_ctrl.in.b_start := FALSE;
						fb_state_entry.i16_next_step := BEREIT;
					END_IF
				END_IF

			BESTUECKZELLE_1720:
			(*-----------------------Weiterschaltbedingungen----------------------------*)
				IF wt_transport_beladen_1720.st_ctrl.out.b_fertig THEN
					wt_transport_beladen_1720.st_ctrl.in.b_start := FALSE;
					fb_state_entry.i16_next_step := BEREIT;
				END_IF
		END_CASE

(*=======================================================*)
	FEHLER:
		IF fb_state_entry.E THEN
			st_ctrl_out.b_fehler := TRUE;
			fb_ton_quitt.IN := FALSE;
			a_foerderband_wt_transport := FALSE;
			wt_transport_beladen.st_ctrl.in.b_stop := TRUE;
			wt_transport_beladen_achse_1700.st_ctrl.in.b_stop  := TRUE;
			wt_transport_warteposition_1700.st_ctrl.in.b_stop  := TRUE;
			wt_transport_abgabe.st_ctrl.in.b_stop := TRUE;
			wt_transport_warteposition_1720.st_ctrl.in.b_stop := TRUE;
			wt_transport_beladen_1720.st_ctrl.in.b_stop := TRUE;
			wt_transport_beladen.st_ctrl.in.b_quitt := FALSE;
			wt_transport_beladen_achse_1700.st_ctrl.in.b_quitt  := FALSE;
			wt_transport_warteposition_1700.st_ctrl.in.b_quitt  := FALSE;
			wt_transport_abgabe.st_ctrl.in.b_quitt := FALSE;
			wt_transport_warteposition_1720.st_ctrl.in.b_quitt := FALSE;
			wt_transport_beladen_1720.st_ctrl.in.b_quitt := FALSE;

			EtherCatDiag[1].st_ctrl_in.b_quitt := FALSE;
			EtherCatDiag[2].st_ctrl_in.b_quitt := FALSE;
			EtherCatDiag[3].st_ctrl_in.b_quitt := FALSE;
			EtherCatDiag[4].st_ctrl_in.b_quitt := FALSE;

			fb_ton_ueberstrom_foerderbaender.IN := FALSE;
		END_IF

		(*-----------------------Weiterschaltbedingungen----------------------------*)
		IF st_ctrl_in.b_quitt AND NOT fb_state_entry.E THEN
			st_ctrl_out.b_fehler := FALSE;
			wt_transport_beladen.st_ctrl.in.b_quitt := TRUE;
			wt_transport_beladen_achse_1700.st_ctrl.in.b_quitt  := TRUE;
			wt_transport_warteposition_1700.st_ctrl.in.b_quitt  := TRUE;
			wt_transport_abgabe.st_ctrl.in.b_quitt := TRUE;
			wt_transport_warteposition_1720.st_ctrl.in.b_quitt := TRUE;
			wt_transport_beladen_1720.st_ctrl.in.b_quitt := TRUE;
			wt_transport_beladen.st_ctrl.in.b_stop := FALSE;
			wt_transport_beladen_achse_1700.st_ctrl.in.b_stop  := FALSE;
			wt_transport_warteposition_1700.st_ctrl.in.b_stop  := FALSE;
			wt_transport_abgabe.st_ctrl.in.b_stop := FALSE;
			wt_transport_warteposition_1720.st_ctrl.in.b_stop := FALSE;
			wt_transport_beladen_1720.st_ctrl.in.b_stop := FALSE;

			EtherCatDiag[1].st_ctrl_in.b_quitt := TRUE;
			EtherCatDiag[2].st_ctrl_in.b_quitt := TRUE;
			EtherCatDiag[3].st_ctrl_in.b_quitt := TRUE;
			EtherCatDiag[4].st_ctrl_in.b_quitt := TRUE;
			fb_ton_quitt.IN := TRUE;
		END_IF

		IF fb_ton_quitt.Q THEN
			fb_ton_quitt.IN := FALSE;
			fb_state_entry.i16_next_step := INIT;
		END_IF

(*=======================================================*)
	STOP:
		IF fb_state_entry.E THEN
			fb_ton_quitt.IN := FALSE;
			a_foerderband_wt_transport := FALSE;
			wt_transport_beladen.st_ctrl.in.b_stop := TRUE;
			wt_transport_beladen_achse_1700.st_ctrl.in.b_stop  := TRUE;
			wt_transport_warteposition_1700.st_ctrl.in.b_stop  := TRUE;
			wt_transport_abgabe.st_ctrl.in.b_stop := TRUE;
			wt_transport_warteposition_1720.st_ctrl.in.b_stop := TRUE;
			wt_transport_beladen_1720.st_ctrl.in.b_stop := TRUE;
			wt_transport_beladen.st_ctrl.in.b_quitt := FALSE;
			wt_transport_beladen_achse_1700.st_ctrl.in.b_quitt  := FALSE;
			wt_transport_warteposition_1700.st_ctrl.in.b_quitt  := FALSE;
			wt_transport_abgabe.st_ctrl.in.b_quitt := FALSE;
			wt_transport_warteposition_1720.st_ctrl.in.b_quitt := FALSE;
			wt_transport_beladen_1720.st_ctrl.in.b_quitt := FALSE;

			EtherCatDiag[1].st_ctrl_in.b_quitt := FALSE;
			EtherCatDiag[2].st_ctrl_in.b_quitt := FALSE;
			EtherCatDiag[3].st_ctrl_in.b_quitt := FALSE;
			EtherCatDiag[4].st_ctrl_in.b_quitt := FALSE;
		END_IF

		(*-----------------------Weiterschaltbedingungen----------------------------*)
		IF st_ctrl_in.b_quitt AND NOT fb_state_entry.E THEN
			fb_ton_quitt.IN := TRUE;
			wt_transport_beladen.st_ctrl.in.b_stop := FALSE;
			wt_transport_beladen_achse_1700.st_ctrl.in.b_stop  := FALSE;
			wt_transport_warteposition_1700.st_ctrl.in.b_stop  := FALSE;
			wt_transport_abgabe.st_ctrl.in.b_stop := FALSE;
			wt_transport_warteposition_1720.st_ctrl.in.b_stop := FALSE;
			wt_transport_beladen_1720.st_ctrl.in.b_stop := FALSE;
			wt_transport_beladen.st_ctrl.in.b_quitt := TRUE;
			wt_transport_beladen_achse_1700.st_ctrl.in.b_quitt  := TRUE;
			wt_transport_warteposition_1700.st_ctrl.in.b_quitt  := TRUE;
			wt_transport_abgabe.st_ctrl.in.b_quitt := TRUE;
			wt_transport_warteposition_1720.st_ctrl.in.b_quitt := TRUE;
			wt_transport_beladen_1720.st_ctrl.in.b_quitt := TRUE;

			EtherCatDiag[1].st_ctrl_in.b_quitt := TRUE;
			EtherCatDiag[2].st_ctrl_in.b_quitt := TRUE;
			EtherCatDiag[3].st_ctrl_in.b_quitt := TRUE;
			EtherCatDiag[4].st_ctrl_in.b_quitt := TRUE;
		END_IF

		IF fb_ton_quitt.Q THEN
			fb_ton_quitt.IN := FALSE;
			fb_state_entry.i16_next_step := INIT;
		END_IF
END_CASE

fb_state_entry(
	i16_next_step:= ,
	i16_pos:= 2,
	s_debugtext:= ,
	E=> ,
	X=> ,
	i16_step=> ,
	i16_last_step=> );

IF st_config.b_config_fertig THEN
	(* Fehlermeldungen ab dem Startindex in das globale Störmeldungsarray schreiben *)
	garr_stoermeldungen[st_config.i16_meld_startindex + 0] := sm_stau_auf_ruecktransport;
	garr_stoermeldungen[st_config.i16_meld_startindex + 1] :=FALSE ;
	garr_stoermeldungen[st_config.i16_meld_startindex + 2] := sm_ueberstrom_foerderbaender;
	garr_stoermeldungen[st_config.i16_meld_startindex + 3] := FALSE;
	garr_stoermeldungen[st_config.i16_meld_startindex + 4] := FALSE;
	garr_stoermeldungen[st_config.i16_meld_startindex + 5] := FALSE;
	garr_stoermeldungen[st_config.i16_meld_startindex + 6] := FALSE;
	garr_stoermeldungen[st_config.i16_meld_startindex + 7] := FALSE;
	garr_stoermeldungen[st_config.i16_meld_startindex + 8] := FALSE;
	garr_stoermeldungen[st_config.i16_meld_startindex + 9] := FALSE;
	garr_stoermeldungen[st_config.i16_meld_startindex + 10] := FALSE;
	garr_stoermeldungen[st_config.i16_meld_startindex + 11] := FALSE;
	garr_stoermeldungen[st_config.i16_meld_startindex + 12] := FALSE;
	garr_stoermeldungen[st_config.i16_meld_startindex + 13] := FALSE;
	garr_stoermeldungen[st_config.i16_meld_startindex + 14] := FALSE;
	garr_stoermeldungen[st_config.i16_meld_startindex + 15] := FALSE;
	garr_stoermeldungen[st_config.i16_meld_startindex + 16] := FALSE;
	garr_stoermeldungen[st_config.i16_meld_startindex + 17] := FALSE;
	garr_stoermeldungen[st_config.i16_meld_startindex + 18] := FALSE;
	garr_stoermeldungen[st_config.i16_meld_startindex + 19] := FALSE;
	
	garr_betriebsmeldungen[st_config.i16_meld_startindex + 0] := bm_einzelfertigung_nach_bandwechsel;
	garr_betriebsmeldungen[st_config.i16_meld_startindex + 1] := FALSE;
	garr_betriebsmeldungen[st_config.i16_meld_startindex + 2] := FALSE;
	garr_betriebsmeldungen[st_config.i16_meld_startindex + 3] := FALSE;
	garr_betriebsmeldungen[st_config.i16_meld_startindex + 4] := FALSE;
	garr_betriebsmeldungen[st_config.i16_meld_startindex + 5] := FALSE;
	garr_betriebsmeldungen[st_config.i16_meld_startindex + 6] := FALSE;
	garr_betriebsmeldungen[st_config.i16_meld_startindex + 7] := FALSE;
	garr_betriebsmeldungen[st_config.i16_meld_startindex + 8] := FALSE;
	garr_betriebsmeldungen[st_config.i16_meld_startindex + 9] := FALSE;
	garr_betriebsmeldungen[st_config.i16_meld_startindex + 10] := FALSE;
	garr_betriebsmeldungen[st_config.i16_meld_startindex + 11] := FALSE;
	garr_betriebsmeldungen[st_config.i16_meld_startindex + 12] := FALSE;
	garr_betriebsmeldungen[st_config.i16_meld_startindex + 13] := FALSE;
	garr_betriebsmeldungen[st_config.i16_meld_startindex + 14] := FALSE;
	garr_betriebsmeldungen[st_config.i16_meld_startindex + 15] := FALSE;
	garr_betriebsmeldungen[st_config.i16_meld_startindex + 16] := FALSE;
	garr_betriebsmeldungen[st_config.i16_meld_startindex + 17] := FALSE;
	garr_betriebsmeldungen[st_config.i16_meld_startindex + 18] := FALSE;
	garr_betriebsmeldungen[st_config.i16_meld_startindex + 19] := FALSE;
END_IF
END_PROGRAM

(* POU Maschine1700/WT Transport/ST_WT_Transport_Warteposition_1700, ST *)
PROGRAM ST_WT_Transport_Warteposition_1700
VAR_INPUT
	st_config								: struct_config;
	st_ctrl_in								: struct_ctrl_in;
	e_station_vorher_in_anforderung			: BOOL := FALSE;
	e_station_vorher_in_abgegeben			: BOOL := FALSE;
END_VAR
VAR_IN_OUT
	st_visu								: struct_visu;
END_VAR
VAR_OUTPUT
	st_ctrl_out							: struct_ctrl_out;
	a_station_vorher_out_erlaubnis			: BOOL := FALSE;
	a_station_vorher_out_angekommen		: BOOL := FALSE;
END_VAR
VAR
	fb_ton_uez							: TON;
	fb_ton_wz							: TON;
	fb_ton_quitt							: TON;
	fb_ton_wt_auf_wartepos				: TON;
	fb_tof_wt_auf_wartepos					: TOF;
	fb_r_trig_start							: R_TRIG;
	fb_r_trig_wartepos						: R_TRIG;
	fb_r_trig_wartepos_verlassen			: R_TRIG;
	fb_state_entry							: ST_StateEntry;
	sm_wt_hat_wartepos_nicht_verlassen	: BOOL := FALSE;
	sm_wt_hat_wartepos_ueberfahren		: BOOL := FALSE;
	bm_warte_anforderung					: BOOL := FALSE;
	bm_warte_wt_an_stopper				: BOOL := FALSE;
	bm_warte_beladepos_frei				: BOOL := FALSE;

	b_helpStartAchse						:BOOL;

	e_wt_auf_wartepos_1700					AT %I* : BOOL;
	e_wt_wartepos_verlassen_1700				AT %I* : BOOL;
END_VAR
(* Zeiten *)
fb_ton_uez(IN:= , PT:= , Q=>  , ET=> );
fb_ton_wz(IN:= , PT:= , Q=> , ET=> );
fb_ton_quitt(IN:= , PT:= t#100ms, Q=> , ET=> );

fb_ton_wt_auf_wartepos(IN:= e_wt_auf_wartepos_1700, PT:= t#200ms, Q=> , ET=> );
fb_tof_wt_auf_wartepos(IN:= e_wt_auf_wartepos_1700, PT:= t#200ms, Q=> , ET=> );

(* Flanken *)
fb_r_trig_wartepos(CLK:= e_wt_auf_wartepos_1700, Q=> );
fb_r_trig_wartepos_verlassen(CLK:= e_wt_wartepos_verlassen_1700, Q=> );
fb_r_trig_start(CLK:= st_ctrl_in.b_start, Q=> );

(* ==================================Toplevel=================================== *)
IF fb_state_entry.i16_next_step > INIT AND fb_state_entry.i16_next_step < FEHLER THEN
	(* Allgemeine Fehler *)
	IF st_ctrl_in.b_stop THEN
		fb_state_entry.i16_next_step := STOP;
	ELSIF zyl_wt_stopper_tisch.st_ctrl.out.b_fehler OR
		zyl_Indexier_Einlauf.st_ctrl.out.b_fehler  THEN
		fb_state_entry.i16_next_step := FEHLER;
	(* Zylinder im Handbetrieb *)
	ELSIF gi16_betriebsart = HAND AND
		st_visu.st_zyl.i16_nr_zyl_im_handbetrieb = zyl_wt_stopper_tisch.fb.st_config.i16_identnummer OR
		st_visu.st_zyl.i16_nr_zyl_im_handbetrieb = zyl_Indexier_Einlauf.fb.st_config.i16_identnummer THEN
			fb_state_entry.i16_next_step := FEHLER;
	END_IF
END_IF

(* ============================Haupt-Schrittkette================================ *)
fb_state_entry(
	i16_next_step:= , 
	i16_pos:= 1,
	s_debugtext:= ,
	E=> ,
	X=> ,
	i16_step=> ,
	i16_last_step=> );

CASE fb_state_entry.i16_step OF
(*=======================================================*)
	INIT_OBJ:
		IF st_config.b_config_fertig THEN
			fb_state_entry.i16_next_step := INIT;
		END_IF

(*=======================================================*)
	INIT:
		IF fb_state_entry.E THEN
			fb_ton_wz.IN := FALSE;
			fb_ton_uez.IN := FALSE;
			fb_ton_quitt.IN := FALSE;
			st_ctrl_out.b_fehler := FALSE;
			st_ctrl_out.b_bereit := FALSE;
			st_ctrl_out.b_fertig := FALSE;
			st_ctrl_out.b_kontroller_start := FALSE;
			zyl_wt_stopper_tisch.st_ctrl.in.b_einfahren := FALSE;
			zyl_wt_stopper_tisch.st_ctrl.in.b_ausfahren := FALSE;
			zyl_Indexier_Einlauf.st_ctrl.in.b_ausfahren := FALSE;
			zyl_Indexier_Einlauf.st_ctrl.in.b_einfahren := FALSE;
			sm_wt_hat_wartepos_nicht_verlassen := FALSE;
			sm_wt_hat_wartepos_ueberfahren := FALSE;
			bm_warte_anforderung := FALSE;
			bm_warte_wt_an_stopper := FALSE;
			bm_warte_beladepos_frei := FALSE;
			a_station_vorher_out_erlaubnis := FALSE;
			a_station_vorher_out_angekommen := FALSE;
			b_helpStartAchse := FALSE;
		END_IF

		(*-----------------------Weiterschaltbedingungen----------------------------*)
		IF st_ctrl_in.b_init THEN
			zyl_wt_stopper_tisch.st_ctrl.in.b_quittieren := FALSE;
			zyl_Indexier_Einlauf.st_ctrl.in.b_quittieren := FALSE;
			fb_state_entry.i16_next_step := 20;
		END_IF

(*=======================================================*)
	20: (* Initialisierung: Prüfe ob WT auf Warteposition *)

		(*-----------------------Weiterschaltbedingungen----------------------------*)
		IF NOT  e_wt_auf_wartepos_1700 THEN
			fb_state_entry.i16_next_step :=  30;
		ELSE
			fb_state_entry.i16_next_step := 40;
		END_IF

(*=======================================================*)
	30: (* Indexierzylinder wieder einfahren und Stopper ausfahren *)
		IF fb_state_entry.E THEN
			zyl_wt_stopper_tisch.st_ctrl.in.b_ausfahren := TRUE;
			zyl_Indexier_Einlauf.st_ctrl.in.b_ausfahren:= TRUE;
		END_IF

		(*-----------------------Weiterschaltbedingungen----------------------------*)
		IF zyl_Indexier_Einlauf.st_ctrl.out.b_ausgefahren THEN
			zyl_Indexier_Einlauf.st_ctrl.in.b_ausfahren:= FALSE;
			zyl_wt_stopper_tisch.st_ctrl.in.b_ausfahren := FALSE;
			fb_state_entry.i16_next_step := BEREIT;
		END_IF

(*=======================================================*)
	40: (*Einlauf Stopper einfahren und WT mit Indexierzylinder fixieren *)

		IF fb_state_entry.E THEN
			zyl_wt_stopper_tisch.st_ctrl.in.b_einfahren := TRUE;
			zyl_Indexier_Einlauf.st_ctrl.in.b_ausfahren:= TRUE;
		END_IF

		(*-----------------------Weiterschaltbedingungen----------------------------*)
		IF 	zyl_wt_stopper_tisch.st_ctrl.out.b_eingefahren AND
			zyl_Indexier_Einlauf.st_ctrl.out.b_ausgefahren AND
			transport_wt_achse.NcToPlc.ActPos <
			gst_datensatz.st_md.st_md_transport_wt_achse.lr_startposition + 0.1 THEN
			zyl_wt_stopper_tisch.st_ctrl.in.b_einfahren := FALSE;
			zyl_Indexier_Einlauf.st_ctrl.in.b_ausfahren:= FALSE;
			fb_state_entry.i16_next_step := 50;
		END_IF

(*=======================================================*)
	50: (*Einlauf Stopper einfahren und WT mit Indexierzylinder fixieren *)

		IF fb_state_entry.E THEN
			zyl_Indexier_Einlauf.st_ctrl.in.b_einfahren:= TRUE;
		END_IF

		(*-----------------------Weiterschaltbedingungen----------------------------*)
		IF 	zyl_Indexier_Einlauf.st_ctrl.out.b_eingefahren THEN
			zyl_Indexier_Einlauf.st_ctrl.in.b_einfahren:= FALSE;
			fb_state_entry.i16_next_step := BEREIT;
		END_IF

(*=======================================================*)
	BEREIT:	(* Warte auf Start von Kontroller *)
		IF fb_state_entry.E THEN
			st_ctrl_out.b_bereit := TRUE;
			st_ctrl_out.b_fertig := TRUE;
		END_IF

		(*-----------------------Weiterschaltbedingungen----------------------------*)
		IF st_config.b_station_aktiv OR st_config.b_station_in_simulation THEN
			(* WT Transport aktiv oder in Simulation *)
			IF st_ctrl_in.b_start THEN
			(* WT Transport gestartet *)
				st_ctrl_out.b_fertig := FALSE;
				fb_state_entry.i16_next_step := 110;
			END_IF
		END_IF

(*=======================================================*)
	110: (* Statische WT-Abfrage auf Warteposition nach der Initialisierung *)
		IF fb_state_entry.E THEN
			st_ctrl_out.b_kontroller_start := TRUE;
		END_IF

		IF NOT e_station_vorher_in_abgegeben THEN
			a_station_vorher_out_angekommen := FALSE;
		END_IF

		(*-----------------------Weiterschaltbedingungen----------------------------*)
		IF e_wt_auf_wartepos_1700 THEN
			st_ctrl_out.b_kontroller_start := FALSE;
			fb_state_entry.i16_next_step := 135;
		ELSE	(* Kein WT da, deshalb einen holen *)
			st_ctrl_out.b_kontroller_start := FALSE;
			fb_state_entry.i16_next_step := 120;
		END_IF

(*=======================================================*)
	120: (* Kein WT da -> warte auf Anforderung von vorheriger Station *)
		IF fb_state_entry.E THEN
			st_ctrl_out.b_kontroller_start := TRUE;
			bm_warte_anforderung := TRUE;
		END_IF

		IF NOT e_station_vorher_in_abgegeben THEN
			a_station_vorher_out_angekommen := FALSE;
		END_IF

		(*-----------------------Weiterschaltbedingungen----------------------------*)
		IF e_station_vorher_in_anforderung THEN
			a_station_vorher_out_angekommen := FALSE;
			a_station_vorher_out_erlaubnis := TRUE;
			st_ctrl_out.b_kontroller_start := FALSE;
			bm_warte_anforderung := FALSE;
			fb_state_entry.i16_next_step := 130;
		END_IF

(*=======================================================*)
	130: (* Warte bis WT an Stopper angekommen ist *)
		IF fb_state_entry.E THEN
			st_ctrl_out.b_kontroller_start := TRUE;
			bm_warte_wt_an_stopper := TRUE;
		END_IF

		(*-----------------------Weiterschaltbedingungen----------------------------*)
		IF fb_r_trig_wartepos.Q THEN
			a_station_vorher_out_erlaubnis := FALSE;
			a_station_vorher_out_angekommen := TRUE;
			st_ctrl_out.b_kontroller_start := FALSE;
			fb_ton_uez.IN := FALSE;
			bm_warte_wt_an_stopper := FALSE;
			fb_state_entry.i16_next_step := 131;
		END_IF

(*=======================================================*)
	131: (* Warte kurz *)
			IF fb_state_entry.E THEN
			fb_ton_wz.PT := t#300ms;
			fb_ton_wz.IN := TRUE;
 		END_IF

		(*-----------------------Weiterschaltbedingungen----------------------------*)
		IF fb_ton_wz.Q THEN
			fb_ton_wz.IN := FALSE;
			fb_state_entry.i16_next_step := 132;
		END_IF

(*=======================================================*)
	132: (*Prüfe ob Achse hinten *)

		(*-----------------------Weiterschaltbedingungen----------------------------*)
		IF  ST_WT_Transport_Achse.lr_Achspos_in = gst_datensatz.st_md.st_md_transport_wt_achse.lr_startposition AND
			axis_transport_wt_achse.st_ctrl.out.b_fertig AND
			NOT axis_transport_wt_achse.st_ctrl.out.b_busy  AND
			NOT axis_transport_wt_achse.st_ctrl.in.b_start  THEN
			fb_state_entry.i16_next_step := 135;
		END_IF

(*=======================================================*)
	135: (*Indexierzylinder Warteposition ausfahren *)
		IF fb_state_entry.E THEN
			zyl_Indexier_Einlauf.st_ctrl.in.b_einfahren:= TRUE;
		END_IF

		(*-----------------------Weiterschaltbedingungen----------------------------*)
		IF zyl_Indexier_Einlauf.st_ctrl.out.b_eingefahren THEN
			zyl_Indexier_Einlauf.st_ctrl.in.b_einfahren:= FALSE;
			fb_state_entry.i16_next_step := 140;
		END_IF

(*=======================================================*)
	140: (* WT ist fixiert -> Einlaufstopper einfahren *)
		IF fb_state_entry.E THEN
			zyl_wt_stopper_tisch.st_ctrl.in.b_einfahren := TRUE;
		END_IF

		(*-----------------------Weiterschaltbedingungen----------------------------*)
		IF zyl_wt_stopper_tisch.st_ctrl.out.b_eingefahren THEN
			zyl_wt_stopper_tisch.st_ctrl.in.b_einfahren := FALSE;
			fb_state_entry.i16_next_step := 145;
		END_IF

(*=======================================================*)
	145: (* Warte kurz *)
			IF fb_state_entry.E THEN
			fb_ton_wz.PT := t#200ms;
			fb_ton_wz.IN := TRUE;
 		END_IF

		(*-----------------------Weiterschaltbedingungen----------------------------*)
		IF fb_ton_wz.Q THEN
			fb_ton_wz.IN := FALSE;
			fb_state_entry.i16_next_step := 150;
		END_IF

(*=======================================================*)
	150: (* Hilfsmerker Achse setzen *)

		(*-----------------------Weiterschaltbedingungen----------------------------*)
		b_helpStartAchse := TRUE;
		fb_state_entry.i16_next_step := 165;

(*=======================================================*)
	165:(*Warten bis Achse ausgefahren ist*)

		(*-----------------------Weiterschaltbedingungen----------------------------*)
		IF ST_WT_Transport_Achse.lr_Achspos_in =gst_datensatz.st_md.st_md_transport_wt_achse.lr_wt_uebergabepos AND
			axis_transport_wt_achse.st_ctrl.out.b_fertig AND
			 zyl_wt_zentrierer_tisch.st_ctrl.out.b_ausgefahren  THEN
			b_helpStartAchse := FALSE;
			fb_state_entry.i16_next_step := 170;
		END_IF

(*=======================================================*)
	170: (* Einlaufstopper ausfahren *)
		IF fb_state_entry.E THEN
			zyl_Indexier_Einlauf.st_ctrl.in.b_ausfahren := TRUE;
			zyl_wt_stopper_tisch.st_ctrl.in.b_ausfahren := TRUE;
		END_IF

		(*-----------------------Weiterschaltbedingungen----------------------------*)
		IF zyl_Indexier_Einlauf.st_ctrl.out.b_ausgefahren THEN
			zyl_Indexier_Einlauf.st_ctrl.in.b_ausfahren := FALSE;
			zyl_wt_stopper_tisch.st_ctrl.in.b_ausfahren := FALSE;
			fb_state_entry.i16_next_step := BEREIT;
		END_IF

(*=======================================================*)
	FEHLER:
		IF fb_state_entry.E THEN
			st_ctrl_out.b_fehler := TRUE;
			fb_ton_quitt.IN := FALSE;
			zyl_wt_stopper_tisch.st_ctrl.in.b_quittieren := FALSE;
			zyl_Indexier_Einlauf.st_ctrl.in.b_quittieren := FALSE;

			a_station_vorher_out_erlaubnis := FALSE;
			a_station_vorher_out_angekommen := FALSE;
		END_IF

		(*-----------------------Weiterschaltbedingungen----------------------------*)
		IF st_ctrl_in.b_quitt AND NOT fb_state_entry.E THEN
			st_ctrl_out.b_fehler := FALSE;
			zyl_wt_stopper_tisch.st_ctrl.in.b_quittieren := TRUE;
			zyl_Indexier_Einlauf.st_ctrl.in.b_quittieren := TRUE;

			fb_ton_quitt.IN := TRUE;
		END_IF

		IF fb_ton_quitt.Q THEN
			fb_ton_quitt.IN := FALSE;
			fb_state_entry.i16_next_step := INIT;
		END_IF

(*=======================================================*)
	STOP:
		IF fb_state_entry.E THEN
			fb_ton_quitt.IN := FALSE;
			st_ctrl_out.b_kontroller_start := FALSE;
			zyl_wt_stopper_tisch.st_ctrl.in.b_quittieren := FALSE;
			zyl_Indexier_Einlauf.st_ctrl.in.b_quittieren := FALSE;

			a_station_vorher_out_erlaubnis := FALSE;
			a_station_vorher_out_angekommen := FALSE;
		END_IF

		(*-----------------------Weiterschaltbedingungen----------------------------*)
		IF st_ctrl_in.b_quitt AND NOT fb_state_entry.E THEN
			fb_ton_quitt.IN := TRUE;
			zyl_wt_stopper_tisch.st_ctrl.in.b_quittieren := TRUE;
			zyl_Indexier_Einlauf.st_ctrl.in.b_quittieren := TRUE;

		END_IF

		IF fb_ton_quitt.Q THEN
			fb_ton_quitt.IN := FALSE;
			fb_state_entry.i16_next_step := INIT;
		END_IF
END_CASE

fb_state_entry(
	i16_next_step:= ,
	i16_pos:= 2,
	s_debugtext:= ,
	E=> ,
	X=> ,
	i16_step=> ,
	i16_last_step=> );

IF st_config.b_config_fertig THEN
	(* Fehlermeldungen ab dem Startindex in das globale Störmeldungsarray schreiben *)
	garr_stoermeldungen[st_config.i16_meld_startindex + 0] := sm_wt_hat_wartepos_nicht_verlassen;
	garr_stoermeldungen[st_config.i16_meld_startindex + 1] := sm_wt_hat_wartepos_ueberfahren;
	garr_stoermeldungen[st_config.i16_meld_startindex + 2] := FALSE;
	garr_stoermeldungen[st_config.i16_meld_startindex + 3] := FALSE;
	garr_stoermeldungen[st_config.i16_meld_startindex + 4] := FALSE;
	garr_stoermeldungen[st_config.i16_meld_startindex + 5] := FALSE;
	garr_stoermeldungen[st_config.i16_meld_startindex + 6] := FALSE;
	garr_stoermeldungen[st_config.i16_meld_startindex + 7] := FALSE;
	garr_stoermeldungen[st_config.i16_meld_startindex + 8] := FALSE;
	garr_stoermeldungen[st_config.i16_meld_startindex + 9] := FALSE;
	garr_stoermeldungen[st_config.i16_meld_startindex + 10] := FALSE;
	garr_stoermeldungen[st_config.i16_meld_startindex + 11] := FALSE;
	garr_stoermeldungen[st_config.i16_meld_startindex + 12] := FALSE;
	garr_stoermeldungen[st_config.i16_meld_startindex + 13] := FALSE;
	garr_stoermeldungen[st_config.i16_meld_startindex + 14] := FALSE;
	garr_stoermeldungen[st_config.i16_meld_startindex + 15] := FALSE;
	garr_stoermeldungen[st_config.i16_meld_startindex + 16] := FALSE;
	garr_stoermeldungen[st_config.i16_meld_startindex + 17] := FALSE;
	garr_stoermeldungen[st_config.i16_meld_startindex + 18] := FALSE;
	garr_stoermeldungen[st_config.i16_meld_startindex + 19] := FALSE;
	
	garr_betriebsmeldungen[st_config.i16_meld_startindex + 0] := bm_warte_anforderung;
	garr_betriebsmeldungen[st_config.i16_meld_startindex + 1] := bm_warte_wt_an_stopper;
	garr_betriebsmeldungen[st_config.i16_meld_startindex + 2] := bm_warte_beladepos_frei;
	garr_betriebsmeldungen[st_config.i16_meld_startindex + 3] := FALSE;
	garr_betriebsmeldungen[st_config.i16_meld_startindex + 4] := FALSE;
	garr_betriebsmeldungen[st_config.i16_meld_startindex + 5] := FALSE;
	garr_betriebsmeldungen[st_config.i16_meld_startindex + 6] := FALSE;
	garr_betriebsmeldungen[st_config.i16_meld_startindex + 7] := FALSE;
	garr_betriebsmeldungen[st_config.i16_meld_startindex + 8] := FALSE;
	garr_betriebsmeldungen[st_config.i16_meld_startindex + 9] := FALSE;
	garr_betriebsmeldungen[st_config.i16_meld_startindex + 10] := FALSE;
	garr_betriebsmeldungen[st_config.i16_meld_startindex + 11] := FALSE;
	garr_betriebsmeldungen[st_config.i16_meld_startindex + 12] := FALSE;
	garr_betriebsmeldungen[st_config.i16_meld_startindex + 13] := FALSE;
	garr_betriebsmeldungen[st_config.i16_meld_startindex + 14] := FALSE;
	garr_betriebsmeldungen[st_config.i16_meld_startindex + 15] := FALSE;
	garr_betriebsmeldungen[st_config.i16_meld_startindex + 16] := FALSE;
	garr_betriebsmeldungen[st_config.i16_meld_startindex + 17] := FALSE;
	garr_betriebsmeldungen[st_config.i16_meld_startindex + 18] := FALSE;
	garr_betriebsmeldungen[st_config.i16_meld_startindex + 19] := FALSE;
END_IF
END_PROGRAM

(* POU Gemeinsamkeiten17xx/Achsen/ST_WT_Transport_Achse, ST *)
PROGRAM ST_WT_Transport_Achse
VAR_INPUT
	st_config_achse						: struct_ecd_config;
	st_ctrl_in								: struct_ctrl_in;
	e_steuerung_ein						: BOOL;
	e_ba_mit_bedingungen				: BOOL;
	e_tuere_vorne_offen					: BOOL;
	e_tuere_hinten_offen					: BOOL;
	lr_tmp_Achspos						: LREAL;
	lr_Achspos_in						: LREAL;
	lr_Velo_in							: LREAL;
	enu_cmd_in						: enum_ecd_cmd;
END_VAR
VAR_IN_OUT
	st_visu								: struct_ecd_visu;
END_VAR
VAR_OUTPUT
	st_ctrl_out							: struct_ctrl_out;
END_VAR
VAR
	st_sm						 		: struct_ecd_meldungen;
	st_drive_cmd							: struct_ecd_cmd;
	fb_ton_wz							: TON;
	fb_ton_quitt							: TON;
	fb_ton_wz_disable						: TON;
	fb_r_trig_start							: R_TRIG;
	fb_r_trig_taste_plus					: R_TRIG;
	fb_r_trig_taste_minus					: R_TRIG;
	fb_r_trig_hand_dialog					: R_TRIG;
	fb_axis								: ST_AxisJobCtrl_Motion;
	fb_state_entry							: ST_StateEntry;
	fb_ton_uez							: TON;
	i									: UINT := 0;
	lr_pos_ohneverschiebung			: LREAL;
	fb_r_trig_limit_sensor_positiv			: R_TRIG;
	fb_r_trig_limit_sensor_negativ			: R_TRIG;
	fb_r_trig_skalierungsnocken				: R_TRIG;
	fb_r_trig_nullpunkt_setzen				: R_TRIG;

	i16_aktuelle_anzahl_bestueckungen		: UINT := 0;
	i16_aktuelle_anzahl_leere_schaechte	: UINT := 0;

	b_hand_dialog_aktiv					: BOOL := FALSE;
	sm_kein_nocken_definiert				: BOOL := FALSE;

	st_geschwindigkeiten					: struct_ecd_geschwindigkeiten;
	e_referenz_sensor						AT %I* : BOOL;
	i16_torque							AT %I* : INT;

	lr_decceleration_nothalt				: LREAL;
	lr_decceleration_normal				: LREAL;

END_VAR
(* Zeiten *)
fb_ton_wz(IN:= , PT:= , Q=>  , ET=> );
fb_ton_uez(IN:= , PT:= , Q=>  , ET=> );
fb_ton_quitt(IN:= , PT:= t#100ms, Q=> , ET=> );
fb_ton_wz_disable(IN:= , PT:= t#500ms, Q=> , ET=> );

(* Flanken *)
fb_r_trig_limit_sensor_positiv(CLK:= st_config_achse.b_limitsensor_positiv_vorhanden AND NOT fb_axis.e_limit_sensor_positive, Q=> );
fb_r_trig_limit_sensor_negativ(CLK:= st_config_achse.b_limitsensor_negativ_vorhanden AND NOT fb_axis.e_limit_sensor_negative, Q=> );
fb_r_trig_taste_plus(CLK:= ST_Euchner_Handbedienpult.b_Taste_Plus, Q=> );
fb_r_trig_taste_minus(CLK:= ST_Euchner_Handbedienpult.b_Taste_Minus, Q=> );
fb_r_trig_start(CLK:= st_ctrl_in.b_start, Q=> );
fb_r_trig_skalierungsnocken(CLK:= nockenschaltwerk_bestueckachse.fb.arr_spur[SP_START_SKALIERUNG], Q=> );
fb_r_trig_hand_dialog(CLK:= b_hand_dialog_aktiv, Q=> );
fb_r_trig_nullpunkt_setzen(CLK:=axis_transport_wt_achse.st_visu.b_nullpunkt_setzen);

(* Achse steuern *)
fb_axis(
	e_referenznocken:= ,
	b_refsensor_vorhanden:= st_config_achse.b_refsensor_vorhanden,
	b_limitsensor_positiv_vorhanden:= st_config_achse.b_limitsensor_positiv_vorhanden,
	b_limitsensor_negativ_vorhanden:= st_config_achse.b_limitsensor_negativ_vorhanden,
	i16_achstyp := st_config_achse.i16_achstyp,
	st_position:= ,
	lr_override_vorgabe:= ST_TippTasten.lr_override,
	mc_richtung_modulo:= ,
	mc_richtung_velocity:= ,
	mc_referenzmodus:= ,
	mc_buffermode_axis:= ,
	ui16_soeparam_write_value:= ,
	w_idn:= ,
	i16_nc_parameter_nummer:= ,
	r_wert_nc_write_parameter:= ,
	st_vorgabe_geschwindigkeiten:= st_geschwindigkeiten,
	lr_soll_geschwindigkeit:= ,
	b_bedingung_sls:= NOT e_tuere_vorne_offen OR NOT e_tuere_hinten_offen,
	st_ads_info := ,
	st_eccoe_sdo := ,
	st_masterachse:= transport_wt_achse,
	st_visu_axis:= st_visu,
	st_ecd_cmd:= st_drive_cmd,
	ui16_soeparam_read_value=> ,
	r_wert_nc_read_parameter=> );

(* Achse mit dem Euchner Handbediengerät vorwärts und rückwärts Bewegen*)
IF gi16_betriebsart = HAND AND fb_r_trig_hand_dialog.Q THEN
	fb_state_entry.i16_next_step := HANDRAD;
END_IF

IF gi16_betriebsart = HAND THEN
	(* Button in der Oberfläche zum setzen des Nullpunktes *)
	IF fb_r_trig_nullpunkt_setzen.Q THEN
		fb_state_entry.i16_next_step := NULLPUNKT_SETZEN;
	END_IF
END_IF


(* =======================================Toplevel========================================== *)
(* Starte Inbetriebnahme-Sequenz *)
IF st_ctrl_in.b_gehe_step_ibn THEN
	fb_state_entry.i16_next_step := INBETRIEBNAHME;
END_IF

(* =====Achse wird disabled===== *)
IF (NOT e_steuerung_ein OR NOT e_ba_mit_bedingungen) AND transport_wt_achse.Status.Operational THEN
	st_drive_cmd.enu_cmd := POWER_DISABLE;
END_IF

IF fb_state_entry.i16_next_step > INIT AND fb_state_entry.i16_next_step < FEHLER THEN
	(* =====Fehler vom Achskontroller===== *)
	IF st_drive_cmd.b_job_fehler THEN
		fb_state_entry.i16_next_step := FEHLER;
	END_IF

	IF fb_state_entry.i16_next_step > 35 THEN
		(* Devicefehler *)
		IF transport_wt_achse.Status.Error THEN
			st_sm.b_achsfehler := TRUE;
			fb_state_entry.i16_next_step := FEHLER;
		ELSIF transport_wt_achse.Status.DriveDeviceError THEN
			st_sm.b_devicefehler := TRUE;
			fb_state_entry.i16_next_step := FEHLER;
		END_IF
	END_IF

	IF fb_state_entry.i16_next_step < STOP THEN
		(* =====Achse wird gestoppt===== *)
		IF st_ctrl_in.b_stop THEN
			fb_state_entry.i16_next_step := STOP;
		ELSIF fb_state_entry.i16_next_step < HALT THEN
			(* =====Achse wird angehalten===== *)
			IF st_ctrl_in.b_halt THEN
				fb_state_entry.i16_next_step := HALT;
			END_IF
		END_IF
	END_IF
END_IF

(* ======================================Schrittkette======================================== *)
fb_state_entry(
	i16_next_step:= ,
	i16_pos:= 1,
	E=> ,
	X=> , 
	i16_step=> ,
	i16_last_step=> );

CASE fb_state_entry.i16_step OF
(*=======================================================*)
	INIT_OBJ:
		IF 	st_config_achse.b_config_fertig AND
			gst_datensatz.st_md.b_anwahl_transport_achse THEN
			fb_state_entry.i16_next_step := 1;
		END_IF

(*=======================================================*)
	1:	(* Warte bis NetID´s der Slaves ausgelesen sind *)
		IF fb_state_entry.E THEN
			;
		END_IF

		(*-----------------------Weiterschaltbedingungen----------------------------*)
		IF ST_EthercatDiag.st_ctrl_out.b_fertig THEN
			fb_state_entry.i16_next_step := 2;
		END_IF

(*=======================================================*)
	2:	(* Spezifische NC-Achsparameter auslesen *)
		IF fb_state_entry.E THEN
			fb_axis.i16_nc_parameter_nummer := MaxVelocitySystem;
			st_drive_cmd.enu_cmd := READ_NC_PARAMETER;
		END_IF

		(*-----------------------Weiterschaltbedingungen----------------------------*)
		IF st_drive_cmd.enu_cmd = NO_COMMAND THEN
			st_geschwindigkeiten.lr_auto_max := st_geschwindigkeiten.lr_maximalgeschwindigkeit := fb_axis.r_wert_nc_read_parameter;
			st_geschwindigkeiten.lr_auto_min := 25.0;
			st_geschwindigkeiten.lr_jog := 50;
			fb_state_entry.i16_next_step := 3;
		END_IF

(*=======================================================*)
	3:	(* Spezifische NC-Achsparameter auslesen *)
		IF fb_state_entry.E THEN
			fb_axis.i16_nc_parameter_nummer := MaxAccelerationSystem;
			st_drive_cmd.enu_cmd := READ_NC_PARAMETER;
		END_IF

		(*-----------------------Weiterschaltbedingungen----------------------------*)
		IF st_drive_cmd.enu_cmd = NO_COMMAND THEN
			st_geschwindigkeiten.lr_beschleunigung := fb_axis.r_wert_nc_read_parameter;
			fb_state_entry.i16_next_step := 4;
		END_IF

(*=======================================================*)
	4:	(* Spezifische NC-Achsparameter auslesen *)
		IF fb_state_entry.E THEN
			fb_axis.i16_nc_parameter_nummer := MaxDecelerationSystem;
			st_drive_cmd.enu_cmd := READ_NC_PARAMETER;
		END_IF

		(*-----------------------Weiterschaltbedingungen----------------------------*)
		IF st_drive_cmd.enu_cmd = NO_COMMAND THEN
			st_geschwindigkeiten.lr_verzoegerung := fb_axis.r_wert_nc_read_parameter;
			lr_decceleration_normal := st_geschwindigkeiten.lr_verzoegerung;
			lr_decceleration_nothalt := 200000.0;
			fb_state_entry.i16_next_step := 5;
		END_IF

(*=======================================================*)
	5:	(* Spezifische NC-Achsparameter auslesen *)
		IF fb_state_entry.E THEN
			fb_axis.i16_nc_parameter_nummer := MaxJerk;
			st_drive_cmd.enu_cmd := READ_NC_PARAMETER;
		END_IF

		(*-----------------------Weiterschaltbedingungen----------------------------*)
		IF st_drive_cmd.enu_cmd = NO_COMMAND THEN
			st_geschwindigkeiten.lr_ruck := fb_axis.r_wert_nc_read_parameter;
			fb_state_entry.i16_next_step := 6;
		END_IF

(*=======================================================*)
	6:	(* Konfigurationen der Achse *)
		IF fb_state_entry.E THEN
			fb_axis.st_eccoe_sdo.s_ec_slave_net_id := ST_EthercatDiag.s_ec_slave_net_id[2];
			fb_axis.st_eccoe_sdo.ui16_slave_addr := st_config_achse.ui16_ethercat_adr;
		END_IF

		(*-----------------------Weiterschaltbedingungen----------------------------*)
		fb_state_entry.i16_next_step := FEHLER; (*in Fehler gehen damit die Achsen resetet werden. Sonst steigen die Achsen bei einem TC Restart aus*)

(*=======================================================*)
	INIT:
		IF fb_state_entry.E THEN
			fb_ton_wz.IN := FALSE;
			fb_ton_uez.IN	:= FALSE;
			fb_ton_quitt.IN := FALSE;
			(* Reset Stoermeldungen *)
			st_sm.b_achse_nicht_auf_startpos := FALSE;
			st_sm.b_achsfehler := FALSE;
			st_sm.b_devicefehler := FALSE;
			st_sm.b_keine_verfahrfreigabe := FALSE;
			st_sm.b_ende_skalierungs_nocke := FALSE;
			st_sm.b_ende_camming_nocke := FALSE;
			st_sm.b_skalierung_noch_aktiv := FALSE;
			st_ctrl_out.b_fehler := FALSE;
			st_ctrl_out.b_fertig := FALSE;
			st_ctrl_out.b_busy:=FALSE;


			st_ctrl_out.b_bereit := FALSE;
			st_ctrl_out.b_prebereit := FALSE;
			sm_kein_nocken_definiert := FALSE;

			fb_axis.lr_soll_geschwindigkeit := gst_datensatz.st_md.r_geschwindigkeit_achse_transport;

			st_geschwindigkeiten.lr_verzoegerung := lr_decceleration_normal;
		END_IF

		(*-----------------------Weiterschaltbedingungen----------------------------*)
		IF st_ctrl_in.b_preinit THEN
			fb_state_entry.i16_next_step := 15;
		END_IF

(*=======================================================*)
	15:	(* Reglerfreigabe wegnehmen *)
		IF fb_state_entry.E THEN
			st_drive_cmd.enu_cmd := POWER_DISABLE;
		END_IF

		(*-----------------------Weiterschaltbedingungen----------------------------*)
		IF st_drive_cmd.enu_cmd = NO_COMMAND THEN
			fb_state_entry.i16_next_step := 20;
		END_IF

(*=======================================================*)
	20:	(* Überprüfe Nullpunktverschiebung des Absolutwertgebers auf Korrektheit *)
		IF fb_state_entry.E THEN
			fb_axis.i16_nc_parameter_nummer := AxisEncoderOffset;	(* vom Datentyp MC_AxisParameter *)
			st_drive_cmd.enu_cmd := READ_NC_PARAMETER;
		END_IF

		(*-----------------------Weiterschaltbedingungen----------------------------*)
		IF st_drive_cmd.enu_cmd = NO_COMMAND THEN
			IF fb_axis.r_wert_nc_read_parameter = gst_datensatz.st_md.st_md_transport_wt_achse.lr_nullpunktverschiebung THEN
				fb_state_entry.i16_next_step := 35;	(* Reglerfreigabe setzen *)
			ELSE
				fb_state_entry.i16_next_step := 25;	(* Nullpunktverschiebung schreiben *)
			END_IF
		END_IF

(*=======================================================*)
	25:	(* Nullpunktverschiebung hat sich geändert, deshalb erst Null reinschreiben, um keinen Additionsfehler zu machen, *)
		(* weil der Wert der Verschiebung beim Neustart komplett auf die Achse geschrieben wird *)
		IF fb_state_entry.E THEN
			fb_axis.i16_nc_parameter_nummer := AxisEncoderOffset;
			fb_axis.r_wert_nc_write_parameter := 0.0;
			st_drive_cmd.enu_cmd := WRITE_NC_PARAMETER;
		END_IF

		(*-----------------------Weiterschaltbedingungen----------------------------*)
		IF st_drive_cmd.enu_cmd = NO_COMMAND THEN
			fb_state_entry.i16_next_step := 30;
		END_IF

(*=======================================================*)
	30:	(* Aktuelle Nullpunktverschiebung des Absolutwertgebers an die Achse senden *)
		IF fb_state_entry.E THEN
			fb_axis.i16_nc_parameter_nummer := AxisEncoderOffset;
			fb_axis.r_wert_nc_write_parameter := gst_datensatz.st_md.st_md_transport_wt_achse.lr_nullpunktverschiebung;
			st_drive_cmd.enu_cmd := WRITE_NC_PARAMETER;
		END_IF

		(*-----------------------Weiterschaltbedingungen----------------------------*)
		IF st_drive_cmd.enu_cmd = NO_COMMAND THEN
			fb_state_entry.i16_next_step := 35;
		END_IF

(*=======================================================*)
	35:	(* Reglerfreigabe setzen , Reset wird bei Bedarf automatisch ausgeführt*)
		IF fb_state_entry.E THEN
			st_drive_cmd.enu_cmd := POWER_ENABLE;
		END_IF

		(*-----------------------Weiterschaltbedingungen----------------------------*)
		IF st_drive_cmd.enu_cmd = NO_COMMAND THEN
			fb_state_entry.i16_next_step := 40;
		END_IF

(*=======================================================*)
	40:	(* Nullpunktverschiebung ist geschrieben *)
		IF fb_state_entry.E THEN
			st_ctrl_out.b_prebereit := TRUE;
		END_IF

		(*-----------------------Weiterschaltbedingungen----------------------------*)
		IF st_ctrl_in.b_init THEN
			fb_state_entry.i16_next_step := BEREIT;
		END_IF

(*=======================================================*)
	45: (* Warte auf Startsignal zum Positionieren *)

		(*-----------------------Weiterschaltbedingungen----------------------------*)
		IF st_ctrl_in.b_start THEN
			fb_state_entry.i16_next_step := 50;
		END_IF

(*=======================================================*)
	50: (* Positioniere Achse auf ausgelesene Slaveposition *)
		IF fb_state_entry.E THEN
			fb_axis.st_position.r_soll := ST_Z_Achse.lr_slave_position;
			st_drive_cmd.enu_cmd := MOVE_ABSOLUTE;
		END_IF

		(*-----------------------Weiterschaltbedingungen----------------------------*)
		IF st_drive_cmd.enu_cmd = NO_COMMAND THEN
			fb_state_entry.i16_next_step := 60;
		END_IF

(*=======================================================*)
	60: (* Warte bis WT Transport Achsegekoppelt wurde *)
		IF fb_state_entry.E THEN
			st_ctrl_out.b_fertig := TRUE;
		END_IF

		(*-----------------------Weiterschaltbedingungen----------------------------*)
		IF transport_wt_achse.NcToPlc.CoupleState = 3 THEN
			st_ctrl_out.b_fertig := FALSE;
			fb_state_entry.i16_next_step := BEREIT;
		END_IF

(*=======================================================*)
	BEREIT:
		IF fb_state_entry.E THEN
			st_ctrl_out.b_bereit := TRUE;
		END_IF

		(*-----------------------Weiterschaltbedingungen----------------------------*)
		IF fb_r_trig_start.Q THEN
			st_ctrl_out.b_fertig := FALSE;
			fb_state_entry.i16_next_step := 110;
		END_IF

		IF 	fb_state_entry.X THEN
			st_ctrl_out.b_busy:= TRUE;
		END_IF

(*=======================================================*)
	110:
		(*-----------------------Weiterschaltbedingungen----------------------------*)
		IF 	st_drive_cmd.enu_cmd = NO_COMMAND THEN
			fb_state_entry.i16_next_step := 120;
		END_IF

(*=======================================================*)
	120: (* Positioniere Achse  *)
		IF 	fb_state_entry.E THEN
			fb_axis.st_position.r_soll := lr_Achspos_in ;
			fb_axis.lr_soll_geschwindigkeit:=lr_Velo_in;
			st_drive_cmd.enu_cmd := enu_cmd_in;
		END_IF

		(*-----------------------Weiterschaltbedingungen----------------------------*)
		IF 	st_drive_cmd.enu_cmd = NO_COMMAND THEN
			st_ctrl_out.b_fertig := TRUE;
			fb_state_entry.i16_next_step := BEREIT;
		END_IF

		IF 	fb_state_entry.X THEN
			st_ctrl_out.b_busy:=FALSE;
		END_IF

(*=======================================================*)
	FEHLER:
		IF fb_state_entry.E THEN
			st_ctrl_out.b_fehler := TRUE;
			fb_ton_quitt.IN := FALSE;
		END_IF

		IF  st_ctrl_in.b_stop AND NOT y_achse.Status.HasBeenStopped THEN
			st_drive_cmd.enu_cmd := STOP_AXIS;
		END_IF

		IF st_ctrl_in.b_halt AND y_achse.Status.Moving THEN
			st_drive_cmd.enu_cmd := HALT_AXIS;
			st_geschwindigkeiten.lr_verzoegerung := lr_decceleration_nothalt;
		END_IF

		(*-----------------------Weiterschaltbedingungen----------------------------*)
		IF st_ctrl_in.b_quitt AND NOT fb_state_entry.E THEN
			st_ctrl_out.b_fehler := FALSE;
			st_drive_cmd.enu_cmd := RESET;
			fb_ton_quitt.IN := TRUE;
		END_IF

		IF fb_ton_quitt.Q THEN
			fb_ton_quitt.IN := FALSE;
			fb_state_entry.i16_next_step := INIT;
		END_IF

		IF	NOT gst_datensatz.st_md.b_anwahl_transport_achse THEN
			st_ctrl_out.b_fehler := FALSE;
			fb_state_entry.i16_next_step := INIT_ObJ;
		END_IF

(*=======================================================*)
	STOP:
		IF fb_state_entry.E THEN
			IF y_achse.NcToPlc.CoupleState = 0 THEN
				st_drive_cmd.enu_cmd := STOP_AXIS;
			END_IF
		END_IF

		(*-----------------------Weiterschaltbedingungen----------------------------*)
		IF st_drive_cmd.enu_cmd = NO_COMMAND AND y_achse.Status.NotMoving THEN
			fb_state_entry.i16_next_step := STILLSTAND;
		END_IF

(*=======================================================*)
	STILLSTAND:
		IF fb_state_entry.E THEN
			st_drive_cmd.enu_cmd := POWER_DISABLE;
			fb_ton_quitt.IN := FALSE;
		END_IF

		(*-----------------------Weiterschaltbedingungen----------------------------*)
		IF st_ctrl_in.b_quitt AND NOT fb_state_entry.E THEN
			fb_ton_quitt.IN := TRUE;
		END_IF

		IF fb_ton_quitt.Q THEN
			fb_ton_quitt.IN := FALSE;
			fb_state_entry.i16_next_step := INIT;
		END_IF

(*=======================================================*)
	HALT:
		IF fb_state_entry.E THEN
			IF y_achse.NcToPlc.CoupleState = 0 THEN
				st_drive_cmd.enu_cmd := HALT_AXIS;
				st_geschwindigkeiten.lr_verzoegerung := lr_decceleration_nothalt;
			END_IF
			fb_ton_quitt.IN := FALSE;
		END_IF

		(*-----------------------Weiterschaltbedingungen----------------------------*)
		IF st_ctrl_in.b_quitt AND NOT fb_state_entry.E THEN
			fb_ton_quitt.IN := TRUE;
		END_IF

		IF fb_ton_quitt.Q THEN
			fb_ton_quitt.IN := FALSE;
			fb_state_entry.i16_next_step := INIT;
		END_IF

(*=======================================================*)
	HANDRAD:	(* Überprüfe Nullpunktverschiebung des Absolutwertgebers auf Korrektheit *)
		IF fb_state_entry.E THEN
			st_ctrl_out.b_fehler := TRUE;
			fb_axis.i16_nc_parameter_nummer := AxisEncoderOffset;
			st_drive_cmd.enu_cmd := READ_NC_PARAMETER;
		END_IF

		(*-----------------------Weiterschaltbedingungen----------------------------*)
		IF st_drive_cmd.enu_cmd = NO_COMMAND THEN
			IF fb_axis.r_wert_nc_read_parameter = gst_datensatz.st_md.st_md_transport_wt_achse.lr_nullpunktverschiebung THEN
				fb_state_entry.i16_next_step := 2040;	(* Jogbetrieb *)
			ELSE
				fb_state_entry.i16_next_step := 2010;	(* Reglerfreigabe nehmen und Nullpunktverschiebung schreiben *)
			END_IF
		END_IF

(*=======================================================*)
	2010:	(* Reglerfreigabe wegnehmen , damit Nullpunktverschiebung geschrieben werden kannt*)
		IF fb_state_entry.E THEN
			st_drive_cmd.enu_cmd := POWER_DISABLE;
		END_IF

		(*-----------------------Weiterschaltbedingungen----------------------------*)
		IF st_drive_cmd.enu_cmd = NO_COMMAND THEN
			fb_state_entry.i16_next_step := 2020;
		END_IF

(*=======================================================*)
	2020:	(* Nullpunktverschiebung hat sich geändert, deshalb erst Null reinschreiben, um keinen Additionsfehler zu machen, *)
			(* weil der Wert der Verschiebung beim Neustart komplett auf die Achse geschrieben wird *)
		IF fb_state_entry.E THEN
			fb_axis.i16_nc_parameter_nummer := AxisEncoderOffset;
			fb_axis.r_wert_nc_write_parameter := 0.0;
			st_drive_cmd.enu_cmd := WRITE_NC_PARAMETER;
		END_IF

		(*-----------------------Weiterschaltbedingungen----------------------------*)
		IF st_drive_cmd.enu_cmd = NO_COMMAND THEN
			fb_state_entry.i16_next_step := 2030;
		END_IF

(*=======================================================*)
	2030:	(* Aktuelle Nullpunktverschiebung des Absolutwertgebers an die Achse senden *)
		IF fb_state_entry.E THEN
			fb_axis.i16_nc_parameter_nummer := AxisEncoderOffset;
			fb_axis.r_wert_nc_write_parameter := gst_datensatz.st_md.st_md_transport_wt_achse.lr_nullpunktverschiebung;
			st_drive_cmd.enu_cmd := WRITE_NC_PARAMETER;
		END_IF

		(*-----------------------Weiterschaltbedingungen----------------------------*)
		IF st_drive_cmd.enu_cmd = NO_COMMAND THEN
			fb_state_entry.i16_next_step := 2040;
		END_IF

(*=======================================================*)
	2040:	(* Jogbetrieb *)
		IF fb_state_entry.E THEN
			fb_axis.lr_soll_geschwindigkeit := st_geschwindigkeiten.lr_jog;
		END_IF

		IF ST_Euchner_Handbedienpult.i16_Handrad_delta > 0 THEN
			st_drive_cmd.enu_cmd := JOG_VORWAERTS;
		ELSIF ST_Euchner_Handbedienpult.i16_Handrad_delta < 0 THEN
			st_drive_cmd.enu_cmd := JOG_RUECKWAERTS;
		ELSIF  y_achse.Status.Moving THEN
			st_drive_cmd.enu_cmd := JOG_STOP;
		END_IF

		IF fb_r_trig_taste_plus.Q THEN
			fb_state_entry.i16_next_step := MOTORBREMSE_AUF;
		END_IF
		IF fb_r_trig_taste_minus.Q THEN
			fb_state_entry.i16_next_step := MOTORBREMSE_ZU;
		END_IF

		(*-----------------------Weiterschaltbedingungen----------------------------*)
		IF gi16_betriebsart <> HAND OR NOT b_hand_dialog_aktiv THEN
			fb_state_entry.i16_next_step := 2050;
		END_IF

(*=======================================================*)
	2050:
		IF fb_state_entry.E THEN
			st_drive_cmd.enu_cmd := ABORT;
		END_IF

		(*-----------------------Weiterschaltbedingungen----------------------------*)
		IF st_drive_cmd.enu_cmd = NO_COMMAND THEN
			fb_state_entry.i16_next_step := 2060;
		END_IF

(*=======================================================*)
	2060:
		IF fb_state_entry.E THEN
			fb_axis.w_idn := P_0_IDN + 96;
			fb_axis.ui16_soeparam_write_value := 0;	(* Motorbremse im Automatikbetrieb für reguläres Fahren *)
			st_drive_cmd.enu_cmd := SOE_WRITE_PARAM;
		END_IF

		(*-----------------------Weiterschaltbedingungen----------------------------*)
		IF st_drive_cmd.enu_cmd = NO_COMMAND THEN
			fb_state_entry.i16_next_step := 2070;
		END_IF

(*=======================================================*)
	2070:	(* Reglerfreigabe wegnehmen *)
		IF fb_state_entry.E THEN
			st_drive_cmd.enu_cmd := POWER_DISABLE;
		END_IF

		(*-----------------------Weiterschaltbedingungen----------------------------*)
		IF st_drive_cmd.enu_cmd = NO_COMMAND THEN
			st_ctrl_out.b_fehler := FALSE;
			fb_state_entry.i16_next_step := INIT;
		END_IF

(*=======================================================*)
	MOTORBREMSE_AUF:
		IF fb_state_entry.E THEN
			st_drive_cmd.enu_cmd := ABORT;
		END_IF

		(*-----------------------Weiterschaltbedingungen----------------------------*)
		IF st_drive_cmd.enu_cmd = NO_COMMAND THEN
			fb_state_entry.i16_next_step := 2110;
		END_IF

(*=======================================================*)
	2110:	(* Reglerfreigabe wegnehmen *)
		IF fb_state_entry.E THEN
			st_drive_cmd.enu_cmd := POWER_DISABLE;
		END_IF

		(*-----------------------Weiterschaltbedingungen----------------------------*)
		IF st_drive_cmd.enu_cmd = NO_COMMAND THEN
			fb_state_entry.i16_next_step := 2120;
		END_IF

(*=======================================================*)
	2120:	(* Bremse auf machen *)
		IF fb_state_entry.E THEN
			fb_axis.w_idn := P_0_IDN + 96;
			fb_axis.ui16_soeparam_write_value := 2;
			st_drive_cmd.enu_cmd := SOE_WRITE_PARAM;
		END_IF

		(*-----------------------Weiterschaltbedingungen----------------------------*)
		IF 	st_drive_cmd.enu_cmd = NO_COMMAND AND
			(gi16_betriebsart <> HAND OR
			NOT b_hand_dialog_aktiv OR
			ST_Euchner_Handbedienpult.i16_Handrad_delta > 0)
			THEN
				fb_state_entry.i16_next_step := HANDRAD;
		ELSIF fb_r_trig_taste_minus.Q THEN
			fb_state_entry.i16_next_step := MOTORBREMSE_ZU;
		END_IF

(*=======================================================*)
	MOTORBREMSE_ZU:
		IF fb_state_entry.E THEN
			st_drive_cmd.enu_cmd := ABORT;
		END_IF

		(*-----------------------Weiterschaltbedingungen----------------------------*)
		IF st_drive_cmd.enu_cmd = NO_COMMAND THEN
			fb_state_entry.i16_next_step := 2210;
		END_IF

(*=======================================================*)
	2210:	(* Reglerfreigabe setzen *)
		IF fb_state_entry.E THEN
			st_drive_cmd.enu_cmd := POWER_ENABLE;
		END_IF

		(*-----------------------Weiterschaltbedingungen----------------------------*)
		IF st_drive_cmd.enu_cmd = NO_COMMAND THEN
			fb_state_entry.i16_next_step := 2220;
		END_IF

(*=======================================================*)
	2220:	(* Bremse zu machen *)
		IF fb_state_entry.E THEN
			fb_axis.w_idn := P_0_IDN + 96;
			fb_axis.ui16_soeparam_write_value := 0;
			st_drive_cmd.enu_cmd := SOE_WRITE_PARAM;
		END_IF

		(*-----------------------Weiterschaltbedingungen----------------------------*)
		IF 	st_drive_cmd.enu_cmd = NO_COMMAND AND
			(gi16_betriebsart <> HAND OR
			NOT b_hand_dialog_aktiv OR
			ST_Euchner_Handbedienpult.i16_Handrad_delta > 0)
			THEN
				fb_state_entry.i16_next_step := HANDRAD;
		ELSIF fb_r_trig_taste_plus.Q THEN
			fb_state_entry.i16_next_step := MOTORBREMSE_AUF;
		END_IF

(*=======================================================*)
	NULLPUNKT_SETZEN:
		(* Aktuellen Jog beenden, sonst Probleme beim Softwareendschalter*)
		IF fb_state_entry.E THEN
			st_drive_cmd.enu_cmd := JOG_STOP;
		END_IF

		(*-----------------------Weiterschaltbedingungen----------------------------*)
		IF st_drive_cmd.enu_cmd = NO_COMMAND THEN
			fb_state_entry.i16_next_step := 2505;
		END_IF

(*=======================================================*)
	2505:
		(* 	Lese aktuelle Nullpunkt verschiebung von der Hardware. Der Benutze könnte einen falschen
			Wert eingetragen haben *)
		IF fb_state_entry.E THEN
			fb_axis.i16_nc_parameter_nummer := AxisEncoderOffset;
			st_drive_cmd.enu_cmd := READ_NC_PARAMETER;
		END_IF

		(*-----------------------Weiterschaltbedingungen----------------------------*)
		IF st_drive_cmd.enu_cmd = NO_COMMAND THEN
			gst_datensatz.st_md.st_md_transport_wt_achse.lr_nullpunktverschiebung := fb_axis.r_wert_nc_read_parameter;
			fb_state_entry.i16_next_step := 2510;
		END_IF

(*=======================================================*)
	2510:	(* Nullpunktverschiebung berechnen *)
		IF fb_state_entry.E THEN
			lr_pos_ohneverschiebung := axis_transport_wt_achse.st_visu.lr_position_ist - gst_datensatz.st_md.st_md_transport_wt_achse.lr_nullpunktverschiebung;

			gst_datensatz.st_md.st_md_transport_wt_achse.lr_nullpunktverschiebung := - lr_pos_ohneverschiebung;
		END_IF

		(*-----------------------Weiterschaltbedingungen----------------------------*)
		(* Aktiviere den wert in die Hardware *)
		fb_state_entry.i16_next_step := HANDRAD;

(*=======================================================*)
	INBETRIEBNAHME:	(* Überprüfe Nullpunktverschiebung des Absolutwertgebers auf Korrektheit *)
		IF fb_state_entry.E THEN
			fb_axis.i16_nc_parameter_nummer := AxisEncoderOffset;
			st_drive_cmd.enu_cmd := READ_NC_PARAMETER;
		END_IF

		(*-----------------------Weiterschaltbedingungen----------------------------*)
		IF st_drive_cmd.enu_cmd = NO_COMMAND THEN
			IF fb_axis.r_wert_nc_read_parameter = gst_datensatz.st_md.st_md_transport_wt_achse.lr_nullpunktverschiebung THEN
				fb_state_entry.i16_next_step := 5100;	(* Reversiersequenz*)
			ELSE
				fb_state_entry.i16_next_step := 5010;	(* Reglerfreigabe nehmen und Nullpunktverschiebung schreiben *)
			END_IF
		END_IF

(*=======================================================*)
	5010:	(* Reglerfreigabe wegnehmen, damit Nullpunktverschiebung geschrieben werden kannt*)
		IF fb_state_entry.E THEN
			st_drive_cmd.enu_cmd := POWER_DISABLE;
		END_IF

		(*-----------------------Weiterschaltbedingungen----------------------------*)
		IF st_drive_cmd.enu_cmd = NO_COMMAND THEN
			fb_state_entry.i16_next_step := 5020;
		END_IF

(*=======================================================*)
	5020:	(* Nullpunktverschiebung hat sich geändert, deshalb erst Null reinschreiben, um keinen Additionsfehler zu machen, *)
			(* weil der Wert der Verschiebung beim Neustart komplett auf die Achse geschrieben wird *)
		IF fb_state_entry.E THEN
			fb_axis.i16_nc_parameter_nummer := AxisEncoderOffset;
			fb_axis.r_wert_nc_write_parameter := 0.0;
			st_drive_cmd.enu_cmd := WRITE_NC_PARAMETER;
		END_IF

		(*-----------------------Weiterschaltbedingungen----------------------------*)
		IF st_drive_cmd.enu_cmd = NO_COMMAND THEN
			fb_state_entry.i16_next_step := 5030;
		END_IF

(*=======================================================*)
	5030:	(* Aktuelle Nullpunktverschiebung des Absolutwertgebers an die Achse senden *)
		IF fb_state_entry.E THEN
			fb_axis.i16_nc_parameter_nummer := AxisEncoderOffset;
			fb_axis.r_wert_nc_write_parameter := gst_datensatz.st_md.st_md_transport_wt_achse.lr_nullpunktverschiebung;
			st_drive_cmd.enu_cmd := WRITE_NC_PARAMETER;
		END_IF

		(*-----------------------Weiterschaltbedingungen----------------------------*)
		IF st_drive_cmd.enu_cmd = NO_COMMAND THEN
			fb_state_entry.i16_next_step := 5100;
		END_IF

(*=======================================================*)
	5100:	(* Verfahren der Achse zwischen zwei Punkten zum Testen verschiedener Achsparameter *)
		IF fb_state_entry.E THEN
			fb_axis.lr_soll_geschwindigkeit := st_geschwindigkeiten.lr_jog;
			fb_axis.st_position.lr_ibn_pos_start := 0.0;
			fb_axis.st_position.lr_ibn_pos_ziel := 25.0;
		END_IF

		(*-----------------------Weiterschaltbedingungen----------------------------*)
		IF st_ctrl_in.b_ibn_start THEN
			fb_state_entry.i16_next_step := 5110;
		END_IF

(*=======================================================*)
	5110: (* Fahre Y-Achse auf Startposition *)
(*
		IF fb_state_entry.E THEN
			 fb_axis.st_position.r_soll := fb_axis.st_position.lr_ibn_pos_start;
			st_drive_cmd.enu_cmd := MOVE_ABSOLUTE;
		END_IF

		(*-----------------------Weiterschaltbedingungen----------------------------*)
		IF st_drive_cmd.enu_cmd = NO_COMMAND THEN
			fb_state_entry.i16_next_step := 5120;
		END_IF
*)
		IF fb_state_entry.E THEN
			st_drive_cmd.enu_cmd := POWER_ENABLE;
		END_IF

		(*-----------------------Weiterschaltbedingungen----------------------------*)
		IF st_drive_cmd.enu_cmd = NO_COMMAND THEN
			;
		END_IF

(*=======================================================*)
	5120: (* Pause *)
		IF fb_state_entry.E THEN
			fb_ton_wz.PT := t#1s;
			fb_ton_wz.IN := TRUE;
		END_IF

		(*-----------------------Weiterschaltbedingungen----------------------------*)
		IF fb_ton_wz.Q THEN
			fb_ton_wz.IN := FALSE;
			fb_state_entry.i16_next_step := 5130;
		END_IF

(*=======================================================*)
	5130: (* Fahre Z-Achse auf Zielposition *)
		IF fb_state_entry.E THEN
			 fb_axis.st_position.r_soll := fb_axis.st_position.lr_ibn_pos_ziel;
			st_drive_cmd.enu_cmd := MOVE_ABSOLUTE;
		END_IF

		(*-----------------------Weiterschaltbedingungen----------------------------*)
		IF st_drive_cmd.enu_cmd = NO_COMMAND THEN
			fb_state_entry.i16_next_step := 5140;
		END_IF

(*=======================================================*)
	5140: (* Pause *)
		IF fb_state_entry.E THEN
			fb_ton_wz.PT := t#1s;
			fb_ton_wz.IN := TRUE;
		END_IF

		(*-----------------------Weiterschaltbedingungen----------------------------*)
		IF fb_ton_wz.Q THEN
			fb_ton_wz.IN := FALSE;
			fb_state_entry.i16_next_step := 5100;
		END_IF
END_CASE

fb_state_entry(
	i16_next_step:= , 
	i16_pos:= 2,
	s_debugtext:= ,
	E=> ,
	X=> ,
	i16_step=> ,
	i16_last_step=> );

